(* CODESYS project Tc3_Mc3Ptp.library
   TcLibraryId: Beckhoff Automation GmbH|Tc3_Mc3Ptp|4.0.17.0
   Company: Beckhoff Automation GmbH
   Title: Tc3_Mc3Ptp
   Placeholder: Tc3_Mc3Ptp
   Version: 4.0.17.0

Project tree, tasks and I/O mapping:
  libraries: Tc3_Mc3Base, 4.0.17.0 (Beckhoff Automation GmbH)
  Motion Objects/
    function block AXIS_REF [ST]: FB_init, FB_exit, InitializeWithOid, GetCamming1DOid, GetPtpErrorResettableOid, GetErrorTriggerableOid, GetMaster1DOid, GetMotionObjectOid, GetPhasing1DOid, GetPtpReadWriteParameterOid, GetPtpSetPositionOid, GetPtpSetHomingStateOid, GetPtpTouchProbeOid, Name, Oid
    function block ENCODER_AXIS_REF [ST]: FB_init, FB_exit, GetPtpErrorResettableOid, GetErrorTriggerableOid, GetMaster1DOid, GetPtpReadWriteParameterOid, GetPtpSetPositionOid, GetPtpSetHomingStateOid, GetPtpTouchProbeOid, Name, Oid
    data type AXIS_REF_TOMC
    data type AXIS_REF_TOPLC
    data type ENCODER_AXIS_REF_TOPLC
  Administrative/
    function block MC_Reset [ST]: FB_init, FB_exit
    function block MC_Power [ST]: FB_init, FB_exit
    function block MC_SetOverride [ST]: FB_init, FB_exit
    Status/
      function block MC_ReadActualPosition [ST]: FB_init, FB_exit
      function block MC_ReadActualTorque [ST]: FB_init, FB_exit
      function block MC_ReadActualVelocity [ST]: FB_init, FB_exit
      function block MC_ReadAxisError [ST]: FB_init, FB_exit
      function block MC_ReadStatus [ST]: FB_init, FB_exit
    function block MC_SetPosition [ST]: FB_init, FB_exit
    Parameter/
      function block MC_WriteHardwareParameter [ST]: FB_init, FB_exit
      function block MC_ReadHardwareParameter [ST]: FB_init, FB_exit
      function block MC_ReadParameter [ST]: FB_init, FB_exit
      function block MC_WriteParameter [ST]: FB_init, FB_exit
      function block MC_ReadBoolParameter [ST]: FB_init, FB_exit
      function block MC_WriteBoolParameter [ST]: FB_init, FB_exit
      data type EAxisParameterId
      data type EReadMode
  External Setpoint Generator/
    function block MC_ActivateExternalSetpointGeneration [ST]: FB_init, FB_exit
    function block MC_ExternalSetpointGenerator [ST]: FB_init, FB_reinit, FB_exit, TcAddRef, TcQueryInterface, TcRelease, GetClassId, TcGetObjectId, TcGetObjectName, TcSetObjectId, TcSetObjectName, TcSetObjState, TcGetObjState, TcGetObjPara, TcSetObjPara, TcGetParentObjId, TcSetParentObjId, OnPreparation, OnStartPointInitialization, OnCyclicSetpointGeneration, OnDeactivation
  Discrete Motion/
    function block MC_Halt [ST]: FB_init, FB_exit
    function block MC_MoveAbsolute [ST]: FB_init, FB_exit
    function block MC_MoveModulo [ST]: FB_init, FB_exit
    function block MC_MoveRelative [ST]: FB_init, FB_exit
    function block MC_Stop [ST]: FB_init, FB_exit
    function block MC_WaitForStableActualPosition [ST]: FB_init, FB_exit
    data type EModuloDirection
  Synchronized Motion/
    function block MC_GearIn [ST]: FB_init, FB_exit
    function block MC_GearInPos [ST]: FB_init, FB_exit
    function block MC_PhasingAbsolute [ST]: FB_init, FB_exit
    function block MC_PhasingRelative [ST]: FB_init, FB_exit
    function block MC_HaltPhasing [ST]: FB_init, FB_exit
    data type EGearInPosSyncState
  Continuous Motion/
    function block MC_MoveVelocity [ST]: FB_init, FB_exit
    function block MC_Jog [ST]: FB_init, FB_exit
    data type EJogMode
  Homing/
    function block MC_SetHomingState [ST]: FB_init, FB_exit
    function block MC_Home [ST]: FB_init, FB_exit
    data type EHomingMode
  TouchProbe/
    function block MC_TouchProbe [ST]: FB_init, FB_exit
    function block MC_AbortTrigger [ST]: FB_init, FB_exit
    function block DriveTouchProbeRef [ST]: FB_init, FB_reinit, FB_exit
    function block EncoderTouchProbeRef [ST]: FB_init, FB_reinit, FB_exit
    function block TimestampTouchProbeRef [ST]: FB_init, FB_reinit, FB_exit
    function block BinaryTouchProbeRef [ST]: FB_init, FB_reinit, FB_exit
    function block FixedStopTouchProbeRef [ST]: FB_init, FB_reinit, FB_exit
    data type TouchProbeOptions
    data type ECoeTouchProbeInput
    data type CoeTouchProbeSettings
    data type FixedStopTouchProbeSettings
    data type EIncrementalEncoderTouchProbeSource
    data type IncrementalEncoderTouchProbeSettings
    data type TRIGGER_REF
    data type TouchProbeUnit
  Load Control/
    function block MC_LoadControl [ST]: FB_init, FB_exit
  Types/
    interface Type_PtpErrorResettable: GetPtpErrorResettableOid
    interface Type_PtpReadWriteParameter: GetPtpReadWriteParameterOid
    interface Type_PtpSetPosition: GetPtpSetPositionOid
    interface Type_PtpSetHomingState: GetPtpSetHomingStateOid
    interface Type_PtpTouchProbe: GetPtpTouchProbeOid
  DUTs/
    data type ESource
  Version/
    global variables Global_Version
*)

// Motion Objects/AXIS_REF_TOMC
(* Contains the information of the AXIS_REF passed from PLC to MC. *)
{attribute 'TcIecLibraryType'}
{attribute 'Namespace' := 'Tc3_Mc3Ptp'}
TYPE AXIS_REF_TOMC : 
	STRUCT
		(* Standard data from PLC to MC. *)
		{attribute 'GUID' := '928ACD6D-34F6-4728-BC12-CB3937EB34C2'}
		{attribute 'Namespace' := 'MC'}
		Std : MC.CDT_PLCTOMC_AXIS_STD;
	END_STRUCT
END_TYPE

// Motion Objects/AXIS_REF_TOPLC
(* Contains the information of the AXIS_REF passed from MC to PLC. *)
{attribute 'TcIecLibraryType'}
{attribute 'Namespace' := 'Tc3_Mc3Ptp'}
TYPE AXIS_REF_TOPLC : 
	STRUCT
		(* Reference to standard data from MC to PLC. *)
		{attribute 'TcPointerMapping'}
		{attribute 'GUID' := 'E7BFE865-900F-4F3A-B607-76F75FE96459'}
		{attribute 'Namespace' := 'MC'}
		Std : REFERENCE TO MC.CDT_MCTOPLC_AXIS_STD;
		(* Reference to setpoint data from MC *)
		{attribute 'TcPointerMapping'}
		{attribute 'GUID' := '0B0DBDAE-EDDB-492C-A6B1-EEFFED71DF0D'}
		{attribute 'Namespace' := 'MC'}
		Set : REFERENCE TO MC.CDT_MCTOPLC_AXIS_SET;
		(* Reference to actpoint data from MC *)
		{attribute 'TcPointerMapping'}
		{attribute 'GUID' := 'B6A63539-66D5-4BB4-8876-F4726B259807'}
		{attribute 'Namespace' := 'MC'}
		Act : REFERENCE TO MC.CDT_MCTOPLC_AXIS_ACT;
		 {attribute 'hide'}
		_reserved1 : ARRAY [1..4] OF UINT_8_16;
		(* Reference to modulo positions of a modulo axis *)
		{attribute 'TcPointerMapping'}
		{attribute 'GUID' := 'A44CE81F-76FF-4B9B-9906-BBAF0C1247D2'}
		{attribute 'Namespace' := 'MC'}
		Modulo : REFERENCE TO MC.CDT_MCTOPLC_AXIS_MODULO;
		(* Reference to loadcontrol data from MC *)
		{attribute 'TcPointerMapping'}
		{attribute 'GUID' := 'FAA1A803-EAD7-4A75-B851-39DA12582F94'}
		{attribute 'Namespace' := 'MC'}
		LoadControl : REFERENCE TO MC.CDT_MCTOPLC_AXIS_LOADCONTROL;
		 {attribute 'hide'}
		_reserved2 : ARRAY [1..8] OF UINT_8_16;
		(* Reference to fluidpower data from MC *)
		{attribute 'TcPointerMapping'}
		{attribute 'GUID' := 'ABD7A116-8AB9-4E1A-99C3-07858EE414A0'}
		{attribute 'Namespace' := 'MC'}
		FluidPower : REFERENCE TO MC.CDT_MCTOPLC_AXIS_FLUIDPOWER;
	END_STRUCT
END_TYPE

// Motion Objects/ENCODER_AXIS_REF_TOPLC
(* Contains the information of the ENCODER_AXIS_REF passed from MC to PLC. *)
{attribute 'TcIecLibraryType'}
{attribute 'Namespace' := 'Tc3_Mc3Ptp'}
TYPE ENCODER_AXIS_REF_TOPLC : 
	STRUCT
		(* Reference to standard data from MC to PLC. *)
		{attribute 'TcPointerMapping'}
		{attribute 'GUID' := 'B8555454-C37F-461B-AA7A-1853577E270C'}
		{attribute 'Namespace' := 'MC'}
		Std : REFERENCE TO MC.CDT_MCTOPLC_ENCODER_AXIS_STD;
		(* Reference to actual data from MC. *)
		{attribute 'TcPointerMapping'}
		{attribute 'GUID' := '104567DA-4469-4052-8B31-85248F22B6DF'}
		{attribute 'Namespace' := 'MC'}
		Act : REFERENCE TO MC.CDT_MCTOPLC_ENCODER_AXIS_ACT;
		(* Reference to modulo positions from encoder axis. *)
		{attribute 'TcPointerMapping'}
		{attribute 'GUID' := '7B38ABBA-E075-4ACD-87B2-5F73D822C5F9'}
		{attribute 'Namespace' := 'MC'}
		Modulo : REFERENCE TO MC.CDT_MCTOPLC_ENCODER_AXIS_MODULO;
	END_STRUCT
END_TYPE

// Discrete Motion/EModuloDirection
(* Direction of travel for modulo positioning. *)
{attribute 'TcIecLibraryType'}
{attribute 'Namespace' := 'Tc3_Mc3Ptp'}
{attribute 'strict'}
{attribute 'qualified_only'}
{attribute 'to_string'}
TYPE EModuloDirection : (
	ShortestDistance:=0, 	(* Move in the direction that results in the shortest travel distance. *)
	PositiveDirection:=1, 	(* Always move in the positive direction to reach the target. *)
	NegativeDirection:=2	(* Always move in the negative direction to reach the target. *)
) UINT;
END_TYPE

// Synchronized Motion/EGearInPosSyncState
(* Synchronization state reported by MC_GearInPos for the PhysicalAxis. Combines whether the slave is synchronized to the master with whether the master has already passed its master sync position. Reports 'Waiting' while the slave cannot move yet due to a sync direction restriction. *)
{attribute 'TcIecLibraryType'}
{attribute 'Namespace' := 'Tc3_Mc3Ptp'}
{attribute 'strict'}
{attribute 'qualified_only'}
{attribute 'to_string'}
TYPE EGearInPosSyncState : (
	Invalid:=0, 	(* Default value before the function block has been activated. *)
	Waiting:=1, 	(* The slave cannot start to move yet because the master is moving against the restricted sync direction. *)
	Synchronizing:=2, 	(* The synchronization is not yet complete and the master has not yet passed its master sync position. *)
	SynchronizingAfterMasterSyncPosition:=3, 	(* The synchronization is not yet complete; the master has already passed its master sync position. *)
	InSyncBeforeMasterSyncPosition:=4, 	(* The slave is locked in to the master, but the master has not yet passed its master sync position. *)
	InSync:=5	(* The slave is locked in to the master and the master has passed its master sync position. *)
) UDINT;
END_TYPE

// Continuous Motion/EJogMode
(* Selects the jog operation mode. *)
{attribute 'TcIecLibraryType'}
{attribute 'Namespace' := 'Tc3_Mc3Ptp'}
{attribute 'strict'}
{attribute 'qualified_only'}
{attribute 'to_string'}
TYPE EJogMode : (
	StandardSlow:=1, 	(* Jog at low velocity using the configured slow jog speed. *)
	StandardFast:=2, 	(* Jog at high velocity using the configured fast jog speed. *)
	Continuous:=3, 	(* Jog continuously at the commanded velocity while the jog input is active. *)
	Inching:=4	(* Move a fixed incremental distance for each jog activation. *)
) UINT;
END_TYPE

// Homing/EHomingMode
(* Mode selection for functional configuration of MC_SetHomingState command. *)
{attribute 'TcIecLibraryType'}
{attribute 'Namespace' := 'Tc3_Mc3Ptp'}
{attribute 'qualified_only'}
{attribute 'strict'}
{attribute 'to_string'}
TYPE EHomingMode : (
	ForceIsHomed:=0, 	(* Sets the homing state to homed (IsPositionValid = TRUE) without performing any movement or position change. *)
	ResetIsHomed:=1, 	(* Resets the homing state to not homed (IsPositionValid = FALSE). *)
	ForceIsHomedAtPosition:=2	(* Sets the current position to the specified homing position and marks the axis as homed (IsPositionValid = TRUE). *)
) UDINT;
END_TYPE

// TouchProbe/TouchProbeOptions
(* MC_TouchProbe Options *)
{attribute 'TcIecLibraryType'}
{attribute 'Namespace' := 'Tc3_Mc3Ptp'}
TYPE TouchProbeOptions : 
	STRUCT
		(* Start position from where trigger events are accepted ([PosUnit], included in the position window).
		It can be left as 'Ignore' if no lower limit is desired. Must have value <= WindowLastPosition otherwise. *)
		WindowFirstPosition : LREAL := STRING_TO_LREAL('#Ignore');
		(* Stop position up to where trigger events are accepted ([PosUnit], included in the position window).
		It can be left as 'Ignore' if no upper limit is desired. Must have value >= WindowFirstPosition otherwise.
		 *)
		WindowLastPosition : LREAL := STRING_TO_LREAL('#Ignore');
		(* Calculate RecordedPosition as modulo value. *)
		PositionsAsModuloValues : BOOL := false;
		(* Continuous recording mode *)
		Continuous : BOOL := false;
		 {attribute 'hide'}
		_reserved1 : ARRAY [1..6] OF USINT;
	END_STRUCT
END_TYPE

// TouchProbe/ECoeTouchProbeInput
(* Selection for CoE Drive touch probe input. *)
{attribute 'TcIecLibraryType'}
{attribute 'Namespace' := 'Tc3_Mc3Ptp'}
{attribute 'qualified_only'}
{attribute 'strict'}
{attribute 'to_string'}
TYPE ECoeTouchProbeInput : (
	DriveDefault:=0, 	(* Trigger on the touch probe default input (i.e., the digital input 1/2 mapped to TouchProbe1/TouchProbe2 functionality in the drive). *)
	ZeroImpulse:=1, 	(* Trigger on the main encoder index signal (encoder Z/index). Only valid if the drive exposes the index signal to the touch probe function. *)
	DriveDefined:=2, 	(* Trigger source is defined by object 0x60D0/0x8001 (DS402/MDP742). *)
	ConfiguredInAxis:=255	(* The touch probe input source is configured in the axis (TCOM object). The value specified at the CoeDriveSettings input is ignored. *)
) UDINT;
END_TYPE

// TouchProbe/CoeTouchProbeSettings
(* CoE drive-specific touch probe source settings. *)
{attribute 'TcIecLibraryType'}
{attribute 'Namespace' := 'Tc3_Mc3Ptp'}
TYPE CoeTouchProbeSettings : 
	STRUCT
		(* Input source for touch probe 1. *)
		{attribute 'GUID' := '119F1828-69D6-4F12-9086-EF2FF951D8CC'}
		{attribute 'Namespace' := 'Tc3_Mc3Ptp'}
		TouchProbe1Source : ECoeTouchProbeInput := ECoeTouchProbeInput.ConfiguredInAxis;
		(* Input source for touch probe 2. *)
		{attribute 'GUID' := '119F1828-69D6-4F12-9086-EF2FF951D8CC'}
		{attribute 'Namespace' := 'Tc3_Mc3Ptp'}
		TouchProbe2Source : ECoeTouchProbeInput := ECoeTouchProbeInput.ConfiguredInAxis;
	END_STRUCT
END_TYPE

// TouchProbe/FixedStopTouchProbeSettings
(* Configure up to three thresholds for fixed stop detection (Torque, Velocity, Lag). Enter #Default to use the axis default value, or #Ignore to disable a threshold.
Typical detection criteria: combination of high torque, low velocity, and/or increasing lag. *)
{attribute 'TcIecLibraryType'}
{attribute 'Namespace' := 'Tc3_Mc3Ptp'}
TYPE FixedStopTouchProbeSettings : 
	STRUCT
		(* Threshold for the actual motor torque. If the torque exceeds this value during evaluation, it contributes to a fixed stop decision. Enter #Ignore to disable this threshold. *)
		TorqueThreshold : LREAL := STRING_TO_LREAL('#Default');
		(* Upper limit for the actual axis velocity during evaluation. Fixed stop detection is evaluated only while the absolute velocity is below this value. Enter #Ignore to disable this threshold. *)
		VelocityThreshold : LREAL := STRING_TO_LREAL('#Default');
		(* Threshold for the position following error (command position minus actual position). If the absolute following error exceeds this value during evaluation, it contributes to a fixed stop decision. Enter #Ignore to disable this threshold. *)
		LagThreshold : LREAL := STRING_TO_LREAL('#Default');
	END_STRUCT
END_TYPE

// TouchProbe/EIncrementalEncoderTouchProbeSource
(* Selection for incremental encoder touch probe latch source. *)
{attribute 'TcIecLibraryType'}
{attribute 'Namespace' := 'Tc3_Mc3Ptp'}
{attribute 'qualified_only'}
{attribute 'strict'}
{attribute 'to_string'}
TYPE EIncrementalEncoderTouchProbeSource : (
	LatchC:=0, 	(* Internal latch (encoder C-track / index signal). *)
	LatchExternPositive:=1, 	(* External latch input, capture on rising edge. *)
	LatchExternNegative:=2, 	(* External latch input, capture on falling edge. *)
	ConfiguredInAxis:=255	(* The touch probe latch source is configured in the axis (TCOM object). The value specified at the IncrementalEncoderSettings input is ignored. *)
) UDINT;
END_TYPE

// TouchProbe/IncrementalEncoderTouchProbeSettings
(* Touch probe settings for incremental encoder terminals. *)
{attribute 'TcIecLibraryType'}
{attribute 'Namespace' := 'Tc3_Mc3Ptp'}
TYPE IncrementalEncoderTouchProbeSettings : 
	STRUCT
		(* Latch source override for position capture. *)
		{attribute 'GUID' := 'B9DA70FA-AB67-491F-BE82-1393AA92E6AD'}
		{attribute 'Namespace' := 'Tc3_Mc3Ptp'}
		Source : EIncrementalEncoderTouchProbeSource := EIncrementalEncoderTouchProbeSource.ConfiguredInAxis;
	END_STRUCT
END_TYPE

// TouchProbe/TRIGGER_REF
{attribute 'TcIecLibraryType'}
{attribute 'Namespace' := 'Tc3_Mc3Ptp'}
{attribute 'hide'}
TYPE TRIGGER_REF : 
	STRUCT
		Target : UDINT;
		ProbeId : UINT;
		 {attribute 'hide'}
		_reserved1 : UINT;
		Edge : UDINT;
		 {attribute 'hide'}
		_reserved2 : UDINT;
		{attribute 'GUID' := '18071995-0000-0000-0000-000000000018'}
		ObjId : GLOBAL.PVOID;
		{attribute 'GUID' := '18071995-0000-0000-0000-000000000018'}
		SettingsCoe : GLOBAL.PVOID;
		{attribute 'GUID' := '18071995-0000-0000-0000-000000000018'}
		SettingsFixedStop : GLOBAL.PVOID;
		{attribute 'GUID' := '18071995-0000-0000-0000-000000000018'}
		SettingsIncrementalEncoder : GLOBAL.PVOID;
	END_STRUCT
END_TYPE

// TouchProbe/TouchProbeUnit
(* Contains trigger references for positive and negative edge touch probes. *)
{attribute 'TcIecLibraryType'}
{attribute 'Namespace' := 'Tc3_Mc3Ptp'}
TYPE TouchProbeUnit : 
	STRUCT
		(* Trigger reference for positive edge events. *)
		{attribute 'GUID' := 'CC3262A1-A7A1-46D3-802E-9117404E77E7'}
		{attribute 'Namespace' := 'Tc3_Mc3Ptp'}
		PositiveTrigger : TRIGGER_REF;
		(* Trigger reference for negative edge events. *)
		{attribute 'GUID' := 'CC3262A1-A7A1-46D3-802E-9117404E77E7'}
		{attribute 'Namespace' := 'Tc3_Mc3Ptp'}
		NegativeTrigger : TRIGGER_REF;
	END_STRUCT
END_TYPE

// DUTs/ESource
(* Selects between setpoint and actual value as data source. *)
{attribute 'TcIecLibraryType'}
{attribute 'Namespace' := 'Tc3_Mc3Ptp'}
{attribute 'hide'}
{attribute 'to_string'}
TYPE ESource : (
	SetValue:=0, 	(* Use the commanded setpoint value. *)
	ActualValue:=1	(* Use the measured actual value from the encoder. *)
) UINT;
END_TYPE

// Administrative/Parameter/EAxisParameterId
(* Parameter IDs for reading and writing axis parameters via MC_ReadParameter / MC_WriteParameter (MC_ReadBoolParameter / MC_WriteBoolParameter). *)
{attribute 'TcIecLibraryType'}
{attribute 'Namespace' := 'Tc3_Mc3Ptp'}
{attribute 'strict'}
{attribute 'qualified_only'}
{attribute 'to_string'}
TYPE EAxisParameterId : (
	Invalid:=16#0000000000000000, 
	MaximumVelocity:=16#0000000005093009, 	(* Use MC_ReadParameter, MC_WriteParameter *)
	MaximumAcceleration:=16#000000000509300a, 	(* Use MC_ReadParameter, MC_WriteParameter *)
	MaximumDeceleration:=16#000000000509300b, 	(* Use MC_ReadParameter, MC_WriteParameter *)
	DefaultAcceleration:=16#000000000509300c, 	(* Use MC_ReadParameter, MC_WriteParameter *)
	DefaultDeceleration:=16#000000000509300d, 	(* Use MC_ReadParameter, MC_WriteParameter *)
	DefaultJerk:=16#000000000509300e, 	(* Use MC_ReadParameter, MC_WriteParameter *)
	MaximumJerk:=16#0000000005093015, 	(* Use MC_ReadParameter, MC_WriteParameter *)
	MinimumPosition:=16#0000000005093021, 	(* Use MC_ReadParameter, MC_WriteParameter *)
	MaximumPosition:=16#0000000005093023, 	(* Use MC_ReadParameter, MC_WriteParameter *)
	PositionModulus:=16#0000000005030107, 	(* Use MC_ReadParameter, MC_WriteParameter *)
	PositionModuloToleranceWindow:=16#0000000005030108, 	(* Use MC_ReadParameter, MC_WriteParameter *)
	MaximumPositionLagValue:=16#000000000503011b, 	(* Use MC_ReadParameter, MC_WriteParameter *)
	MaximumPositionLagFilterTime:=16#000000000503011c, 	(* Use MC_ReadParameter, MC_WriteParameter *)
	JogVelocitySlow:=16#000000000503019e, 	(* Use MC_ReadParameter, MC_WriteParameter *)
	JogVelocityFast:=16#000000000503019f, 	(* Use MC_ReadParameter, MC_WriteParameter *)
	MinimumPositionLag:=16#00000000050301a1, 	(* Use MC_ReadParameter, MC_WriteParameter *)
	MaximumPositionLag:=16#00000000050301a2, 	(* Use MC_ReadParameter, MC_WriteParameter *)
	VelocityOverrideFactor:=16#0000000005030231, 	(* Use MC_ReadParameter, MC_WriteParameter *)
	SimulationMode:=16#00000000050300b1, 	(* Use MC_ReadBoolParameter, MC_WriteBoolParameter *)
	IsModuloAxis:=16#0000000005030101, 	(* Use MC_ReadBoolParameter, MC_WriteBoolParameter *)
	PositionLagMonitoringEnabled:=16#000000000503011a, 	(* Use MC_ReadBoolParameter, MC_WriteBoolParameter *)
	PositionLimitEnforcementEnabled:=16#000000000503015d, 	(* Use MC_ReadBoolParameter, MC_WriteBoolParameter *)
	DriveVelocityScalingNumeratorToHardware:=16#0000000105030122, 	(* Use MC_ReadParameter, MC_WriteParameter *)
	DriveVelocityScalingDenominatorToHardware:=16#00000001050301a7, 	(* Use MC_ReadParameter, MC_WriteParameter *)
	DriveTorqueScalingFromHardware:=16#000000010503014f, 	(* Use MC_ReadParameter, MC_WriteParameter *)
	DriveTimeoutForEnableAndReset:=16#000000010503d004, 	(* Use MC_ReadParameter, MC_WriteParameter *)
	DriveActiveHomingOffset:=16#0000000105030224, 	(* Use MC_ReadParameter, MC_WriteParameter *)
	DriveDirectionInverted:=16#00000001050301b2, 	(* Use MC_ReadBoolParameter, MC_WriteBoolParameter *)
	EncoderPositionScalingNumeratorFromHardware:=16#0000000205030103, 	(* Use MC_ReadParameter, MC_WriteParameter *)
	EncoderPositionScalingDenominatorFromHardware:=16#0000000205030104, 	(* Use MC_ReadParameter, MC_WriteParameter *)
	EncoderMountingOffset:=16#0000000205030106, 	(* Use MC_ReadParameter, MC_WriteParameter *)
	EncoderWorkZeroOffset:=16#00000002050301d1, 	(* Use MC_ReadParameter, MC_WriteParameter *)
	EncoderDirectionInverted:=16#00000002050301b2, 	(* Use MC_ReadBoolParameter, MC_WriteBoolParameter *)
	EncoderIsHomed:=16#000000020503d070, 	(* Use MC_ReadBoolParameter, MC_WriteBoolParameter *)
	EncoderIsAbsolutePositionValid:=16#000000020503d071	(* Use MC_ReadBoolParameter, MC_WriteBoolParameter *)
) ULINT;
END_TYPE

// Administrative/Parameter/EReadMode
(* Selects the read operation mode. *)
{attribute 'TcIecLibraryType'}
{attribute 'Namespace' := 'Tc3_Mc3Ptp'}
{attribute 'strict'}
{attribute 'qualified_only'}
{attribute 'to_string'}
TYPE EReadMode : (
	Once:=1, 	(* Read the parameter value once. *)
	Cyclic:=2	(* Read the parameter value cyclically. *)
) UDINT;
END_TYPE

// Version/Global_Version
{attribute 'TcGenerated'}
// This function has been automatically generated from the project information.
VAR_GLOBAL CONSTANT
	{attribute 'const_non_replaced'}
	{attribute 'linkalways'}
	stLibVersion_Tc3_Mc3Ptp : ST_LibVersion := (iMajor := 4, iMinor := 0, iBuild := 17, iRevision := 0, nFlags := 0, sVersion := '4.0.17.0');
	{attribute 'const_non_replaced'}
	{attribute 'linkalways'}
	sLibraryId_Tc3_Mc3Ptp : String := 'Beckhoff Automation GmbH|Tc3_Mc3Ptp|4.0.17.0';
END_VAR

// Motion Objects/AXIS_REF

{attribute 'c++_compatible'}
{attribute 'external_name' := 'AXIS_REF_GUID_931209B0_6FAC_E9BE_F824_23CE2FAA5732'}
{attribute 'TcIecLibraryType'}
(* 
        An MC3 axis used with PLCopen motion control function blocks.
	 *)
FUNCTION_BLOCK AXIS_REF IMPLEMENTS Tc3_Mc3Base.Type_Camming1D, Type_PtpErrorResettable, Tc3_Mc3Base.Type_ErrorTriggerable, Tc3_Mc3Base.Type_Master1D, Tc3_Mc3Base.Type_MotionObject, Tc3_Mc3Base.Type_Phasing1D, Type_PtpReadWriteParameter, Type_PtpSetPosition, Type_PtpSetHomingState, Type_PtpTouchProbe
VAR
END_VAR
VAR_INPUT
	(* Data area for cyclic PLC-to-MC data exchange (mapped to MC axis TcCOM object input process image). *)
	{attribute 'GUID' := '70EBE612-C6D0-4BB5-85F1-59AB9BBF86DE'}
	{attribute 'Namespace' := 'Tc3_Mc3Ptp'}
	PlcToMc AT %Q* : AXIS_REF_TOMC;
	(* Data area for cyclic MC-to-PLC data exchange (mapped to MC axis TcCOM object output process image). *)
	{attribute 'GUID' := '99E83C85-C326-4077-86A5-05990B8F1158'}
	{attribute 'Namespace' := 'Tc3_Mc3Ptp'}
	McToPlc AT %I* : AXIS_REF_TOPLC;
END_VAR
VAR
	{attribute 'hide'}
	_reserved : UDINT;
	 {attribute 'hide'}
	_reserved1 : UINT_0_32;
END_VAR

{attribute 'TcTypeSystem'}

(* Internal method *)
{attribute 'hide'}
METHOD FB_init : BOOL
VAR_INPUT
	(*  if TRUE, the retain variables are initialized (warm start / cold start) *)
	bInitRetains : BOOL;
	(*  if TRUE, the instance afterwards gets moved into the copy code (online change) *)
	bInCopyCode : BOOL;
END_VAR
END_METHOD

{attribute 'TcTypeSystem'}

(* Internal method *)
{attribute 'hide'}
METHOD FB_exit : BOOL
VAR_INPUT
	(*  if TRUE, the exit method is called for exiting an instance that is copied afterwards (online change). *)
	bInCopyCode : BOOL;
END_VAR
END_METHOD

{attribute 'TcTypeSystem'}

(* Internal method to wrap object ID *)
{attribute 'hide'}
METHOD InitializeWithOid
VAR_INPUT
	(* Object ID which is used as an alternative when this is used as master. *)
	{attribute 'GUID' := '18071995-0000-0000-0000-00000000000F'}
	NewOid : GLOBAL.OTCID;
END_VAR
END_METHOD

{attribute 'TcTypeSystem'}

{attribute 'c++_external'}
{attribute 'hide'}
METHOD GetCamming1DOid : GLOBAL.OTCID
END_METHOD

{attribute 'TcTypeSystem'}

{attribute 'c++_external'}
{attribute 'hide'}
METHOD GetPtpErrorResettableOid : GLOBAL.OTCID
END_METHOD

{attribute 'TcTypeSystem'}

{attribute 'c++_external'}
{attribute 'hide'}
METHOD GetErrorTriggerableOid : GLOBAL.OTCID
END_METHOD

{attribute 'TcTypeSystem'}

{attribute 'c++_external'}
{attribute 'hide'}
METHOD GetMaster1DOid : GLOBAL.OTCID
END_METHOD

{attribute 'TcTypeSystem'}

{attribute 'c++_external'}
{attribute 'hide'}
METHOD GetMotionObjectOid : GLOBAL.OTCID
END_METHOD

{attribute 'TcTypeSystem'}

{attribute 'c++_external'}
{attribute 'hide'}
METHOD GetPhasing1DOid : GLOBAL.OTCID
END_METHOD

{attribute 'TcTypeSystem'}

{attribute 'c++_external'}
{attribute 'hide'}
METHOD GetPtpReadWriteParameterOid : GLOBAL.OTCID
END_METHOD

{attribute 'TcTypeSystem'}

{attribute 'c++_external'}
{attribute 'hide'}
METHOD GetPtpSetPositionOid : GLOBAL.OTCID
END_METHOD

{attribute 'TcTypeSystem'}

{attribute 'c++_external'}
{attribute 'hide'}
METHOD GetPtpSetHomingStateOid : GLOBAL.OTCID
END_METHOD

{attribute 'TcTypeSystem'}

{attribute 'c++_external'}
{attribute 'hide'}
METHOD GetPtpTouchProbeOid : GLOBAL.OTCID
END_METHOD

{attribute 'TcTypeSystem'}

	(* Returns the configured name of the axis. *)
{attribute 'monitoring' := 'call'}
	PROPERTY Name : STRING(255)
GET
END_GET
END_PROPERTY

{attribute 'TcTypeSystem'}

	(* Returns the TcCOM object ID of the axis. *)
{attribute 'monitoring' := 'call'}
	PROPERTY Oid : GLOBAL.OTCID
GET
END_GET
END_PROPERTY

END_FUNCTION_BLOCK

// Types/Type_PtpErrorResettable
(* Type for a motion control object whose errors can be reset (e. g. supported by AXIS_REF). *)
{attribute 'Namespace' := 'Tc3_Mc3Ptp'}
{attribute 'c++_compatible'}
INTERFACE Type_PtpErrorResettable

{attribute 'TcTypeSystem'}
{attribute 'c++_compatible'}
{attribute 'minimal_input_size' := '4'}
{attribute 'pack_mode' := '4'}
{attribute 'hide'}
METHOD GetPtpErrorResettableOid : GLOBAL.OTCID
END_METHOD

END_INTERFACE

// Types/Type_PtpReadWriteParameter
(* Type for a motion control object that supports parameter read/write access (e.g. supported by AXIS_REF and ENCODER_AXIS_REF). *)
{attribute 'Namespace' := 'Tc3_Mc3Ptp'}
{attribute 'c++_compatible'}
INTERFACE Type_PtpReadWriteParameter

{attribute 'TcTypeSystem'}
{attribute 'c++_compatible'}
{attribute 'minimal_input_size' := '4'}
{attribute 'pack_mode' := '4'}
{attribute 'hide'}
METHOD GetPtpReadWriteParameterOid : GLOBAL.OTCID
END_METHOD

END_INTERFACE

// Motion Objects/ENCODER_AXIS_REF

{attribute 'c++_compatible'}
{attribute 'external_name' := 'ENCODER_AXIS_REF_GUID_E0F25744_2FAD_E888_F942_A6877B2D0404'}
{attribute 'TcIecLibraryType'}
(* 
        An MC3 encoder axis used with PLCopen motion control function blocks.
	 *)
FUNCTION_BLOCK ENCODER_AXIS_REF IMPLEMENTS Type_PtpErrorResettable, Tc3_Mc3Base.Type_ErrorTriggerable, Tc3_Mc3Base.Type_Master1D, Type_PtpReadWriteParameter, Type_PtpSetPosition, Type_PtpSetHomingState, Type_PtpTouchProbe
VAR
END_VAR
VAR_INPUT
	(* Data area for cyclic MC-to-PLC data exchange (mapped to MC encoder axis TcCOM object output process image). *)
	{attribute 'GUID' := 'B5C6D7E8-F9A0-4B1C-2D3E-4F5A6B7C8D9E'}
	{attribute 'Namespace' := 'Tc3_Mc3Ptp'}
	McToPlc AT %I* : ENCODER_AXIS_REF_TOPLC;
END_VAR

{attribute 'TcTypeSystem'}

(* Internal method *)
{attribute 'hide'}
METHOD FB_init : BOOL
VAR_INPUT
	(*  if TRUE, the retain variables are initialized (warm start / cold start) *)
	bInitRetains : BOOL;
	(*  if TRUE, the instance afterwards gets moved into the copy code (online change) *)
	bInCopyCode : BOOL;
END_VAR
END_METHOD

{attribute 'TcTypeSystem'}

(* Internal method *)
{attribute 'hide'}
METHOD FB_exit : BOOL
VAR_INPUT
	(*  if TRUE, the exit method is called for exiting an instance that is copied afterwards (online change). *)
	bInCopyCode : BOOL;
END_VAR
END_METHOD

{attribute 'TcTypeSystem'}

{attribute 'c++_external'}
{attribute 'hide'}
METHOD GetPtpErrorResettableOid : GLOBAL.OTCID
END_METHOD

{attribute 'TcTypeSystem'}

{attribute 'c++_external'}
{attribute 'hide'}
METHOD GetErrorTriggerableOid : GLOBAL.OTCID
END_METHOD

{attribute 'TcTypeSystem'}

{attribute 'c++_external'}
{attribute 'hide'}
METHOD GetMaster1DOid : GLOBAL.OTCID
END_METHOD

{attribute 'TcTypeSystem'}

{attribute 'c++_external'}
{attribute 'hide'}
METHOD GetPtpReadWriteParameterOid : GLOBAL.OTCID
END_METHOD

{attribute 'TcTypeSystem'}

{attribute 'c++_external'}
{attribute 'hide'}
METHOD GetPtpSetPositionOid : GLOBAL.OTCID
END_METHOD

{attribute 'TcTypeSystem'}

{attribute 'c++_external'}
{attribute 'hide'}
METHOD GetPtpSetHomingStateOid : GLOBAL.OTCID
END_METHOD

{attribute 'TcTypeSystem'}

{attribute 'c++_external'}
{attribute 'hide'}
METHOD GetPtpTouchProbeOid : GLOBAL.OTCID
END_METHOD

{attribute 'TcTypeSystem'}

	(* Returns the configured name of the encoder axis. *)
{attribute 'monitoring' := 'call'}
	PROPERTY Name : STRING(255)
GET
END_GET
END_PROPERTY

{attribute 'TcTypeSystem'}

	(* Returns the TcCOM object ID of the encoder axis. *)
{attribute 'monitoring' := 'call'}
	PROPERTY Oid : GLOBAL.OTCID
GET
END_GET
END_PROPERTY

END_FUNCTION_BLOCK

// Types/Type_PtpSetPosition
(* Type for a motion control object that supports setting position (e. g. supported by AXIS_REF). *)
{attribute 'Namespace' := 'Tc3_Mc3Ptp'}
{attribute 'c++_compatible'}
INTERFACE Type_PtpSetPosition

{attribute 'TcTypeSystem'}
{attribute 'c++_compatible'}
{attribute 'minimal_input_size' := '4'}
{attribute 'pack_mode' := '4'}
{attribute 'hide'}
METHOD GetPtpSetPositionOid : GLOBAL.OTCID
END_METHOD

END_INTERFACE

// Types/Type_PtpSetHomingState
(* Type for a motion control object that supports setting the homing state (e. g. supported by AXIS_REF and ENCODER_AXIS_REF). *)
{attribute 'Namespace' := 'Tc3_Mc3Ptp'}
{attribute 'c++_compatible'}
INTERFACE Type_PtpSetHomingState

{attribute 'TcTypeSystem'}
{attribute 'c++_compatible'}
{attribute 'minimal_input_size' := '4'}
{attribute 'pack_mode' := '4'}
{attribute 'hide'}
METHOD GetPtpSetHomingStateOid : GLOBAL.OTCID
END_METHOD

END_INTERFACE

// Types/Type_PtpTouchProbe
(* Type for a motion control object that supports touch probe commands (e. g. supported by AXIS_REF and ENCODER_AXIS_REF). *)
{attribute 'Namespace' := 'Tc3_Mc3Ptp'}
{attribute 'c++_compatible'}
INTERFACE Type_PtpTouchProbe

{attribute 'TcTypeSystem'}
{attribute 'c++_compatible'}
{attribute 'minimal_input_size' := '4'}
{attribute 'pack_mode' := '4'}
{attribute 'hide'}
METHOD GetPtpTouchProbeOid : GLOBAL.OTCID
END_METHOD

END_INTERFACE

// Administrative/MC_Reset

{attribute 'c++_compatible'}
{attribute 'external_name' := 'MC_Reset_GUID_C09B70BA_4675_EE3C_E76C_41428371BC38'}
{attribute 'TcIecLibraryType'}
{attribute 'hide_all_locals'}
(* 
		This function block resets all motion object-related errors and transitions the motion object out of state ErrorStop.<br/>
		The resulting state is Disabled, if no Enable is requested for the motion object (e.g. via MC_Power).<br/>
		It results in DiscreteMotion, if the motion object has a closed control loop and a controlled error reaction is still ongoing.<br/>
		Otherwise, Standstill is the resulting state. This function block does not affect the output of motion function block instances.
	 *)
FUNCTION_BLOCK MC_Reset
VAR_INPUT
	(* Interface pointer to the object on which the command should be performed (e.g. Axis, Linear Mover). *)
	{attribute 'GUID' := '871876B3-D74D-4115-B995-E302FD1B35FF'}
	{attribute 'Namespace' := 'Tc3_Mc3Ptp'}
	Axis : Type_PtpErrorResettable;
	(* Trigger the command with rising edge. *)
	Execute : BOOL;
END_VAR
VAR_OUTPUT
	(* Potential axis and/or drive error has been reset. State Standstill, Disabled or DiscreteMotion is reached. *)
	Done : BOOL;
	(* Function block is not finished and new output values are to be expected. *)
	Busy : BOOL;
	(* Error occurred within function block. *)
	Error : BOOL;
	(* Error identifier *)
	ErrorId : UDINT;
END_VAR
VAR
	 {attribute 'hide'}
	_reserved1 : UINT_0_32;
	 {attribute 'hide'}
	_reserved2 : ARRAY [1..20] OF UINT_8_16;
	 {attribute 'hide'}
	_reserved3 : ARRAY [1..28] OF USINT;
END_VAR

{attribute 'TcTypeSystem'}

(* Internal method *)
{attribute 'hide'}
METHOD FB_init : BOOL
VAR_INPUT
	(*  if TRUE, the retain variables are initialized (warm start / cold start) *)
	bInitRetains : BOOL;
	(*  if TRUE, the instance afterwards gets moved into the copy code (online change) *)
	bInCopyCode : BOOL;
END_VAR
END_METHOD

{attribute 'TcTypeSystem'}

(* Internal method *)
{attribute 'hide'}
METHOD FB_exit : BOOL
VAR_INPUT
	(*  if TRUE, the exit method is called for exiting an instance that is copied afterwards (online change). *)
	bInCopyCode : BOOL;
END_VAR
END_METHOD

END_FUNCTION_BLOCK

// Administrative/MC_Power

{attribute 'c++_compatible'}
{attribute 'external_name' := 'MC_Power_GUID_DFCA01AC_8B4E_E5B3_DB59_8C7638CFE540'}
{attribute 'TcIecLibraryType'}
{attribute 'hide_all_locals'}
(* 
		This function block controls the power stage (on or off).
	 *)
FUNCTION_BLOCK MC_Power
VAR_IN_OUT
	(* Reference to the axis *)
	{attribute 'GUID' := '931209B0-6FAC-E9BE-F824-23CE2FAA5732'}
	{attribute 'Namespace' := 'Tc3_Mc3Ptp'}
	Axis : AXIS_REF;
END_VAR
VAR_INPUT
	(* General software enable for the axis *)
	Enable : BOOL;
	(* Feed enable in positive direction. Only effective if Enable = TRUE *)
	EnablePositive : BOOL := false;
	(* Feed enable in negative direction. Only effective if Enable = TRUE *)
	EnableNegative : BOOL := false;
END_VAR
VAR_OUTPUT
	(* Axis is ready for motion commands. *)
	Status : BOOL;
	(* Error occurred within function block or axis already signaling an error. *)
	Error : BOOL;
END_VAR
VAR
	 {attribute 'hide'}
	_reserved1 : ARRAY [1..3] OF USINT;
END_VAR
VAR_OUTPUT
	(* Error identifier of function block or axis *)
	ErrorId : UDINT;
END_VAR
VAR
	 {attribute 'hide'}
	_reserved2 : UINT_0_32;
END_VAR

{attribute 'TcTypeSystem'}

(* Internal method *)
{attribute 'hide'}
METHOD FB_init : BOOL
VAR_INPUT
	(*  if TRUE, the retain variables are initialized (warm start / cold start) *)
	bInitRetains : BOOL;
	(*  if TRUE, the instance afterwards gets moved into the copy code (online change) *)
	bInCopyCode : BOOL;
END_VAR
END_METHOD

{attribute 'TcTypeSystem'}

(* Internal method *)
{attribute 'hide'}
METHOD FB_exit : BOOL
VAR_INPUT
	(*  if TRUE, the exit method is called for exiting an instance that is copied afterwards (online change). *)
	bInCopyCode : BOOL;
END_VAR
END_METHOD

END_FUNCTION_BLOCK

// Administrative/MC_SetOverride

{attribute 'c++_compatible'}
{attribute 'external_name' := 'MC_SetOverride_GUID_EC43C2CD_0650_E2EE_F82C_55B33981EAD6'}
{attribute 'TcIecLibraryType'}
{attribute 'hide_all_locals'}
(* 
	This function block sets the velocity override factor that is applied to movement commands of the axis.
	The override factor does not apply to movement in the synchronized motion state (e.g. movement induced by MC_GearIn, MC_GearInPos, ...).
	 *)
FUNCTION_BLOCK MC_SetOverride
VAR_IN_OUT
	(* Reference to the axis *)
	{attribute 'GUID' := '931209B0-6FAC-E9BE-F824-23CE2FAA5732'}
	{attribute 'Namespace' := 'Tc3_Mc3Ptp'}
	Axis : AXIS_REF;
END_VAR
VAR_INPUT
	(* Write the velocity override factor continuously while Enable = TRUE. *)
	Enable : BOOL;
END_VAR
VAR
	 {attribute 'hide'}
	_reserved1 : ARRAY [1..7] OF USINT;
END_VAR
VAR_INPUT
	(* Applies to commanded velocities. Valid range is [0,1]. Use STRING_TO_LREAL('#Ignore') to NOT overwrite the previous value. *)
	VelocityFactor : LREAL := 1.0;
END_VAR
VAR
	 {attribute 'hide'}
	_reserved2 : ARRAY [1..8] OF USINT;
END_VAR
VAR_OUTPUT
	(* The commanded override is set. *)
	Enabled : BOOL;
	(* Error occurred within function block. *)
	Error : BOOL;
END_VAR
VAR
	 {attribute 'hide'}
	_reserved3 : UINT;
END_VAR
VAR_OUTPUT
	(* Error identifier *)
	ErrorId : UDINT;
END_VAR

{attribute 'TcTypeSystem'}

(* Internal method *)
{attribute 'hide'}
METHOD FB_init : BOOL
VAR_INPUT
	(*  if TRUE, the retain variables are initialized (warm start / cold start) *)
	bInitRetains : BOOL;
	(*  if TRUE, the instance afterwards gets moved into the copy code (online change) *)
	bInCopyCode : BOOL;
END_VAR
END_METHOD

{attribute 'TcTypeSystem'}

(* Internal method *)
{attribute 'hide'}
METHOD FB_exit : BOOL
VAR_INPUT
	(*  if TRUE, the exit method is called for exiting an instance that is copied afterwards (online change). *)
	bInCopyCode : BOOL;
END_VAR
END_METHOD

END_FUNCTION_BLOCK

// Synchronized Motion/MC_GearIn

{attribute 'c++_compatible'}
{attribute 'external_name' := 'MC_GearIn_GUID_D7A1F00E_B353_E326_E653_99E98F4ECC09'}
{attribute 'TcIecLibraryType'}
{attribute 'hide_all_locals'}
(* 
		This function block commands a ratio between the velocity of the slave and master axis.
	 *)
FUNCTION_BLOCK MC_GearIn
VAR_INPUT
	(* Reference to the master axis *)
	{attribute 'Namespace' := 'Tc3_Mc3Base'}
	Master : Tc3_Mc3Base.Type_Master1D;
	(* Reference to the slave axis *)
	{attribute 'GUID' := '931209B0-6FAC-E9BE-F824-23CE2FAA5732'}
	{attribute 'Namespace' := 'Tc3_Mc3Ptp'}
	Slave : REFERENCE TO AXIS_REF;
	(* Trigger the command with rising edge. *)
	Execute : BOOL;
END_VAR
VAR
	 {attribute 'hide'}
	_reserved1 : UINT_24_56;
END_VAR
VAR_INPUT
	(* Gear ratio numerator *)
	RatioNumerator : LREAL := 1.0;
	(* Gear ratio denominator *)
	RatioDenominator : UDINT := 1;
END_VAR
VAR
END_VAR
VAR_INPUT
	(* Maximum slave acceleration ([PosUnit]/s^2, positive) *)
	Acceleration : LREAL := STRING_TO_LREAL('#Default');
	(* Maximum slave deceleration ([PosUnit]/s^2, positive) *)
	Deceleration : LREAL := STRING_TO_LREAL('#Default');
	(* Maximum slave jerk ([PosUnit]/s^3, positive) *)
	Jerk : LREAL := STRING_TO_LREAL('#Default');
	(* Chronological sequence of the command *)
	{attribute 'Namespace' := 'Tc3_Mc3Base'}
	BufferMode : Tc3_Mc3Base.EBufferMode := Tc3_Mc3Base.EBufferMode.Aborting;
	(* Reaction if an error occurs in the master while this command is active. *)
	{attribute 'Namespace' := 'Tc3_Mc3Base'}
	ReactionToMasterError : Tc3_Mc3Base.EReactionToMasterError := Tc3_Mc3Base.EReactionToMasterError.TriggerSlaveError;
	(* Reaction if an error occurs in the slave while this command is active. *)
	{attribute 'Namespace' := 'Tc3_Mc3Base'}
	ReactionToSlaveError : Tc3_Mc3Base.EReactionToSlaveError := Tc3_Mc3Base.EReactionToSlaveError.TriggerMasterError;
END_VAR
VAR
END_VAR
VAR_OUTPUT
	(* Synchronization established *)
	InGear : BOOL;
	(* Function block is not finished and new output values are to be expected. *)
	Busy : BOOL;
	(* Function block has active control on the axis. *)
	Active : BOOL;
	(* Command is aborted by another command. *)
	CommandAborted : BOOL;
	(* Error occurred within function block. *)
	Error : BOOL;
END_VAR
VAR
	 {attribute 'hide'}
	_reserved2 : USINT;
END_VAR
VAR_OUTPUT
	(* Error identifier *)
	ErrorId : UDINT;
	(* Master is in error state. *)
	MasterHasError : BOOL;
END_VAR
VAR
	 {attribute 'hide'}
	_reserved3 : UINT_24_56;
	 {attribute 'hide'}
	_reserved4 : ARRAY [1..40] OF UINT_8_16;
	 {attribute 'hide'}
	_reserved5 : ARRAY [1..8] OF USINT;
END_VAR

{attribute 'TcTypeSystem'}

(* Internal method *)
{attribute 'hide'}
METHOD FB_init : BOOL
VAR_INPUT
	(*  if TRUE, the retain variables are initialized (warm start / cold start) *)
	bInitRetains : BOOL;
	(*  if TRUE, the instance afterwards gets moved into the copy code (online change) *)
	bInCopyCode : BOOL;
END_VAR
END_METHOD

{attribute 'TcTypeSystem'}

(* Internal method *)
{attribute 'hide'}
METHOD FB_exit : BOOL
VAR_INPUT
	(*  if TRUE, the exit method is called for exiting an instance that is copied afterwards (online change). *)
	bInCopyCode : BOOL;
END_VAR
END_METHOD

END_FUNCTION_BLOCK

// Synchronized Motion/MC_GearInPos

{attribute 'c++_compatible'}
{attribute 'pack_mode' := '1'}
{attribute 'external_name' := 'MC_GearInPos_GUID_4134C37A_5B73_E5EF_D747_25D272B58ACA'}
{attribute 'TcIecLibraryType'}
{attribute 'hide_all_locals'}
(* 
		This function block commands a gear ratio between the position of the slave and master axes
		from the synchronization point onwards.
	 *)
FUNCTION_BLOCK MC_GearInPos
VAR_INPUT
	(* Reference to the master axis *)
	{attribute 'Namespace' := 'Tc3_Mc3Base'}
	Master : Tc3_Mc3Base.Type_Master1D;
	(* Reference to the slave axis *)
	{attribute 'GUID' := '931209B0-6FAC-E9BE-F824-23CE2FAA5732'}
	{attribute 'Namespace' := 'Tc3_Mc3Ptp'}
	Slave : REFERENCE TO AXIS_REF;
	(* Trigger the command with rising edge. *)
	Execute : BOOL;
END_VAR
VAR
	 {attribute 'hide'}
	_reserved1 : UINT_24_56;
END_VAR
VAR_INPUT
	(* Gear ratio numerator *)
	RatioNumerator : LREAL := 1.0;
	(* Gear ratio denominator *)
	RatioDenominator : UDINT := 1;
END_VAR
VAR
	 {attribute 'hide'}
	_reserved2 : UDINT;
END_VAR
VAR_INPUT
	(* Position of master axis where master and slave axis are synchronized. *)
	MasterSyncPosition : LREAL := STRING_TO_LREAL('#Invalid');
	(* Position of slave axis where master and slave axis are synchronized. *)
	SlaveSyncPosition : LREAL := STRING_TO_LREAL('#Invalid');
	(* Maximum velocity during synchronization ([PosUnit]/s, positive) *)
	Velocity : LREAL := STRING_TO_LREAL('#Maximum');
	(* Maximum acceleration during synchronization ([PosUnit]/s^2, positive) *)
	Acceleration : LREAL := STRING_TO_LREAL('#Default');
	(* Maximum deceleration during synchronization ([PosUnit]/s^2, positive) *)
	Deceleration : LREAL := STRING_TO_LREAL('#Default');
	(* Maximum jerk during synchronization ([PosUnit]/s^3, positive) *)
	Jerk : LREAL := STRING_TO_LREAL('#Default');
	(* Chronological sequence of the command *)
	{attribute 'Namespace' := 'Tc3_Mc3Base'}
	BufferMode : Tc3_Mc3Base.EBufferMode := Tc3_Mc3Base.EBufferMode.Aborting;
	(* Reaction if an error occurs in the master while this command is active. *)
	{attribute 'Namespace' := 'Tc3_Mc3Base'}
	ReactionToMasterError : Tc3_Mc3Base.EReactionToMasterError := Tc3_Mc3Base.EReactionToMasterError.TriggerSlaveError;
	(* Reaction if an error occurs in the slave while this command is active. *)
	{attribute 'Namespace' := 'Tc3_Mc3Base'}
	ReactionToSlaveError : Tc3_Mc3Base.EReactionToSlaveError := Tc3_Mc3Base.EReactionToSlaveError.TriggerMasterError;
END_VAR
VAR
END_VAR
VAR_INPUT
	(* Allowed directions for establishing initial synchronization *)
	{attribute 'Namespace' := 'Tc3_Mc3Base'}
	AllowedSlaveSyncDirections : Tc3_Mc3Base.ESyncDirection := Tc3_Mc3Base.ESyncDirection.TowardsSlaveSyncPosition;
END_VAR
VAR
END_VAR
VAR_OUTPUT
	(* Synchronization started *)
	{attribute 'hide'}
	StartSync : BOOL;
	(* True if SyncState == InSync (slave coupled to the master AND master has passed its master sync position). *)
	InSync : BOOL;
END_VAR
VAR
	 {attribute 'hide'}
	_reserved3 : UINT;
END_VAR
VAR_OUTPUT
	(* Synchronization state. See EGearInPosSyncState for details. *)
	{attribute 'GUID' := 'C1F4A2D8-3B7E-4D5F-9A2C-8E6B1F0D4A93'}
	{attribute 'Namespace' := 'Tc3_Mc3Ptp'}
	SyncState : EGearInPosSyncState;
	(* Function block is not finished and new output values are to be expected. *)
	Busy : BOOL;
	(* Function block has active control on the axis. *)
	Active : BOOL;
	(* Command is aborted by another command. *)
	CommandAborted : BOOL;
	(* Error occurred within function block. *)
	Error : BOOL;
	(* Error identifier *)
	ErrorId : UDINT;
	(* Master is in error state. *)
	MasterHasError : BOOL;
END_VAR
VAR
	 {attribute 'hide'}
	_reserved4 : UINT_24_56;
	 {attribute 'hide'}
	_reserved5 : ARRAY [1..32] OF UINT_8_16;
	 {attribute 'hide'}
	_reserved6 : ARRAY [1..24] OF USINT;
END_VAR

{attribute 'TcTypeSystem'}

(* Internal method *)
{attribute 'hide'}
METHOD FB_init : BOOL
VAR_INPUT
	(*  if TRUE, the retain variables are initialized (warm start / cold start) *)
	bInitRetains : BOOL;
	(*  if TRUE, the instance afterwards gets moved into the copy code (online change) *)
	bInCopyCode : BOOL;
END_VAR
END_METHOD

{attribute 'TcTypeSystem'}

(* Internal method *)
{attribute 'hide'}
METHOD FB_exit : BOOL
VAR_INPUT
	(*  if TRUE, the exit method is called for exiting an instance that is copied afterwards (online change). *)
	bInCopyCode : BOOL;
END_VAR
END_METHOD

END_FUNCTION_BLOCK

// Administrative/MC_SetPosition

{attribute 'c++_compatible'}
{attribute 'external_name' := 'MC_SetPosition_GUID_14AA4E3B_998A_E180_F419_69B3FBB763F2'}
{attribute 'TcIecLibraryType'}
{attribute 'hide_all_locals'}
(* 
		This function block shifts the coordinate system of an axis by manipulating both the setpoint position as well as the
		actual position of an axis with the same value without any movement caused (Re-calibration with same following error).
		This can be used for instance for a reference situation.
	 *)
FUNCTION_BLOCK MC_SetPosition
VAR_INPUT
	(* Reference to the axis *)
	{attribute 'GUID' := 'F2078C57-FA2D-4316-A502-6E36DE58DC4A'}
	{attribute 'Namespace' := 'Tc3_Mc3Ptp'}
	Axis : Type_PtpSetPosition;
	(* Trigger the command with rising edge. *)
	Execute : BOOL;
END_VAR
VAR
	 {attribute 'hide'}
	_reserved1 : ARRAY [1..7] OF USINT;
END_VAR
VAR_INPUT
	(* New position value ([PosUnit]) or distance if Relative = TRUE *)
	Position : LREAL := STRING_TO_LREAL('#Invalid');
	(* Shift axis position by value *)
	Relative : BOOL := false;
	(* Resets position lag to zero. *)
	ClearPositionLag : BOOL;
END_VAR
VAR_OUTPUT
	(* Position has new value. *)
	Done : BOOL;
	(* Function block is not finished and new output values are to be expected. *)
	Busy : BOOL;
	(* Error occurred within function block. *)
	Error : BOOL;
END_VAR
VAR
	 {attribute 'hide'}
	_reserved2 : ARRAY [1..3] OF USINT;
END_VAR
VAR_OUTPUT
	(* Error identifier *)
	ErrorId : UDINT;
END_VAR
VAR
	 {attribute 'hide'}
	_reserved3 : UINT_0_32;
	 {attribute 'hide'}
	_reserved4 : ARRAY [1..20] OF UINT_8_16;
	 {attribute 'hide'}
	_reserved5 : ARRAY [1..32] OF USINT;
END_VAR

{attribute 'TcTypeSystem'}

(* Internal method *)
{attribute 'hide'}
METHOD FB_init : BOOL
VAR_INPUT
	(*  if TRUE, the retain variables are initialized (warm start / cold start) *)
	bInitRetains : BOOL;
	(*  if TRUE, the instance afterwards gets moved into the copy code (online change) *)
	bInCopyCode : BOOL;
END_VAR
END_METHOD

{attribute 'TcTypeSystem'}

(* Internal method *)
{attribute 'hide'}
METHOD FB_exit : BOOL
VAR_INPUT
	(*  if TRUE, the exit method is called for exiting an instance that is copied afterwards (online change). *)
	bInCopyCode : BOOL;
END_VAR
END_METHOD

END_FUNCTION_BLOCK

// External Setpoint Generator/MC_ActivateExternalSetpointGeneration

{attribute 'c++_compatible'}
{attribute 'external_name' := 'MC_ActivateExternalSetpointGeneration_GUID_F01B1D76_5347_ED41_C01F_C4347FBFE6A0'}
{attribute 'TcIecLibraryType'}
{attribute 'hide_all_locals'}
(* 
		This function block activates external setpoint generation.
		Setpoints are generated by a function block, which is called through the ITcMcExternalSetpointGenerator interface from the MC context.
		Additionally custom startup data can be passed through the generator.
	 *)
FUNCTION_BLOCK MC_ActivateExternalSetpointGeneration
VAR_IN_OUT
	(* Reference to the axis *)
	{attribute 'GUID' := '931209B0-6FAC-E9BE-F824-23CE2FAA5732'}
	{attribute 'Namespace' := 'Tc3_Mc3Ptp'}
	Axis : AXIS_REF;
END_VAR
VAR_INPUT
	(* Trigger the command with rising edge. *)
	Execute : BOOL;
END_VAR
VAR
	 {attribute 'hide'}
	_reserved1 : UINT_24_56;
END_VAR
VAR_INPUT
	(* Function block that implements (cyclic) methods for external setpoint generation *)
	{attribute 'GUID' := 'EF828E0B-69F0-4553-9DFF-4817D2FD6510'}
	ExternalSetpointGenerator : GLOBAL.ITcMcExternalSetpointGenerator;
	(* Allow the calling task to differ from the MC task (MET task). When TRUE, ensure compatible update rates and safe data access in the ITcMcExternalSetpointGenerator methods. *)
	AllowOtherContext : BOOL := false;
	(* Trigger error on inconsistent setpoint values (position, velocity, acceleration) if EnableDynamicChecks = TRUE. *)
	EnableDynamicChecks : BOOL := true;
END_VAR
VAR
	 {attribute 'hide'}
	_reserved2 : UINT_16_48;
END_VAR
VAR_INPUT
	(* Invocation identifier, passed through to the external setpoint generator. Can be used to distinguish multiple activations of the same generator, or to pass custom data (e.g. a pointer). *)
	{attribute 'GUID' := '18071995-0000-0000-0000-000000000073'}
	InvokeId : GLOBAL.XWORD := 0;
	(* Chronological sequence of the command *)
	{attribute 'Namespace' := 'Tc3_Mc3Base'}
	BufferMode : Tc3_Mc3Base.EBufferMode := Tc3_Mc3Base.EBufferMode.Aborting;
END_VAR
VAR_OUTPUT
	(* Function block is not finished and new output values are to be expected. *)
	Busy : BOOL;
	(* Function block has active control on the axis. *)
	Active : BOOL;
	(* Command is aborted by another command. *)
	CommandAborted : BOOL;
	(* Error occurred within function block. *)
	Error : BOOL;
END_VAR
VAR
	 {attribute 'hide'}
	_reserved3 : UINT;
END_VAR
VAR_OUTPUT
	(* Error identifier *)
	ErrorId : UDINT;
END_VAR
VAR
	 {attribute 'hide'}
	_reserved4 : UINT_0_32;
	 {attribute 'hide'}
	_reserved5 : ARRAY [1..32] OF UINT_8_16;
	 {attribute 'hide'}
	_reserved6 : ARRAY [1..24] OF USINT;
END_VAR

{attribute 'TcTypeSystem'}

(* Internal method *)
{attribute 'hide'}
METHOD FB_init : BOOL
VAR_INPUT
	(*  if TRUE, the retain variables are initialized (warm start / cold start) *)
	bInitRetains : BOOL;
	(*  if TRUE, the instance afterwards gets moved into the copy code (online change) *)
	bInCopyCode : BOOL;
END_VAR
END_METHOD

{attribute 'TcTypeSystem'}

(* Internal method *)
{attribute 'hide'}
METHOD FB_exit : BOOL
VAR_INPUT
	(*  if TRUE, the exit method is called for exiting an instance that is copied afterwards (online change). *)
	bInCopyCode : BOOL;
END_VAR
END_METHOD

END_FUNCTION_BLOCK

// External Setpoint Generator/MC_ExternalSetpointGenerator

{attribute 'c++_compatible'}
{attribute 'external_name' := 'MC_ExternalSetpointGenerator_GUID_395BF1E9_74A7_EC7E_CCDB_6EE07212C52C'}
{attribute 'TcIecLibraryType'}
{attribute 'no_explicit_call' :='do not call this POU directly'}
{attribute 'c++_compatible'}
{attribute 'hide_all_locals'}
(* 
	This function block provides the API to implement an external setpoint generator from the PLC environment.<br/>
The included callback methods are called from MC task context.<br/>
At least the OnCyclicSetpointGeneration method must be implemented.<br/>
<br/>
Requirements for deriving function block:<br/>
- The function block must implement ITcMcExternalSetpointGenerator interface.<br/>
- The function block and all overridden ITcMcExternalSetpointGenerator methods must have {attribute 'c++_compatible'}.<br/>
- The function block must override FB_init.<br/>
<br/>
Notes:<br/>
For online change compatibility the function block must have a FB_reinit method, in which MC_ExternalSetpointGenerator.FB_reinit() is called.
	 *)
FUNCTION_BLOCK ABSTRACT MC_ExternalSetpointGenerator IMPLEMENTS GLOBAL.ITComObject, GLOBAL.ITcMcExternalSetpointGenerator
VAR
	reserved : ARRAY [1..64] OF BYTE;
END_VAR

{attribute 'TcTypeSystem'}

(* (Internal method.) Initializes the function block with the object name. *)
METHOD FB_init : BOOL
VAR_INPUT
	(*  if TRUE, the retain variables are initialized (warm start / cold start) *)
	bInitRetains : BOOL;
	(*  if TRUE, the instance afterwards gets moved into the copy code (online change) *)
	bInCopyCode : BOOL;
	{attribute 'GUID' := '18071995-0000-0000-0000-000100000050'}
	sObjectName : STRING;
END_VAR
END_METHOD

{attribute 'TcTypeSystem'}

(* Internal method *)
METHOD FB_reinit : BOOL
END_METHOD

{attribute 'TcTypeSystem'}

(* Internal method *)
METHOD FB_exit : BOOL
VAR_INPUT
	(*  if TRUE, the exit method is called for exiting an instance that is copied afterwards (online change). *)
	bInCopyCode : BOOL;
END_VAR
END_METHOD

{attribute 'TcTypeSystem'}

(* Internal method *)
{attribute 'c++_compatible'}
{attribute 'hide'}
METHOD FINAL TcAddRef : UDINT
END_METHOD

{attribute 'TcTypeSystem'}

(* Internal method *)
{attribute 'c++_compatible'}
{attribute 'c++_external'}
{attribute 'hide'}
METHOD FINAL TcQueryInterface : GLOBAL.HRESULT
VAR_INPUT
	{attribute 'GUID' := '18071995-0000-0000-0000-000000000025'}
	iid : REFERENCE TO GLOBAL.IID;
	{attribute 'GUID' := '18071995-0000-0000-0000-000000000018'}
	pipItf : POINTER TO GLOBAL.PVOID;
END_VAR
END_METHOD

{attribute 'TcTypeSystem'}

(* Internal method *)
{attribute 'c++_compatible'}
{attribute 'c++_external'}
{attribute 'hide'}
METHOD FINAL TcRelease : UDINT
END_METHOD

{attribute 'TcTypeSystem'}

{attribute 'c++_compatible'}
{attribute 'c++_external'}
{attribute 'hide'}
METHOD FINAL GetClassId : GLOBAL.HRESULT
VAR_INPUT
	{attribute 'GUID' := '18071995-0000-0000-0000-000000000024'}
	classId : REFERENCE TO GLOBAL.CLSID;
END_VAR
END_METHOD

{attribute 'TcTypeSystem'}

{attribute 'c++_compatible'}
{attribute 'c++_external'}
{attribute 'hide'}
METHOD FINAL TcGetObjectId : GLOBAL.HRESULT
VAR_INPUT
	{attribute 'GUID' := '18071995-0000-0000-0000-00000000000F'}
	objId : REFERENCE TO GLOBAL.OTCID;
END_VAR
END_METHOD

{attribute 'TcTypeSystem'}

{attribute 'c++_compatible'}
{attribute 'c++_external'}
{attribute 'hide'}
METHOD FINAL TcGetObjectName : GLOBAL.HRESULT
VAR_INPUT
	objName : POINTER TO SINT;
	nameLen : UDINT;
END_VAR
END_METHOD

{attribute 'TcTypeSystem'}

{attribute 'c++_compatible'}
{attribute 'c++_external'}
{attribute 'hide'}
METHOD FINAL TcSetObjectId : GLOBAL.HRESULT
VAR_INPUT
	{attribute 'GUID' := '18071995-0000-0000-0000-00000000000F'}
	objId : GLOBAL.OTCID;
END_VAR
END_METHOD

{attribute 'TcTypeSystem'}

{attribute 'c++_compatible'}
{attribute 'c++_external'}
{attribute 'hide'}
METHOD FINAL TcSetObjectName : GLOBAL.HRESULT
VAR_INPUT
	objName : POINTER TO SINT;
END_VAR
END_METHOD

{attribute 'TcTypeSystem'}

{attribute 'c++_compatible'}
{attribute 'c++_external'}
{attribute 'hide'}
METHOD FINAL TcSetObjState : GLOBAL.HRESULT
VAR_INPUT
	{attribute 'GUID' := '18071995-0000-0000-0000-000000000061'}
	state : GLOBAL.TCOM_STATE;
	{attribute 'GUID' := '00000030-0000-0000-E000-000000000064'}
	ipSrv : GLOBAL.ITComObjectServer;
	{attribute 'GUID' := '8ADAFA6E-467B-49AA-BC54-CA235CC732A9'}
	pInitData : POINTER TO GLOBAL.TComInitDataHdr;
END_VAR
END_METHOD

{attribute 'TcTypeSystem'}

{attribute 'c++_compatible'}
{attribute 'c++_external'}
{attribute 'hide'}
METHOD FINAL TcGetObjState : GLOBAL.HRESULT
VAR_INPUT
	{attribute 'GUID' := '18071995-0000-0000-0000-000000000061'}
	pState : POINTER TO GLOBAL.TCOM_STATE;
END_VAR
END_METHOD

{attribute 'TcTypeSystem'}

{attribute 'c++_compatible'}
{attribute 'c++_external'}
{attribute 'hide'}
METHOD FINAL TcGetObjPara : GLOBAL.HRESULT
VAR_INPUT
	{attribute 'GUID' := '18071995-0000-0000-0000-00000000001C'}
	pid : GLOBAL.PTCID;
	nData : REFERENCE TO UDINT;
	{attribute 'GUID' := '18071995-0000-0000-0000-000000000018'}
	pData : REFERENCE TO GLOBAL.PVOID;
	{attribute 'GUID' := '18071995-0000-0000-0000-00000000001D'}
	pgp : GLOBAL.PTCGP := 0;
END_VAR
END_METHOD

{attribute 'TcTypeSystem'}

{attribute 'c++_compatible'}
{attribute 'c++_external'}
{attribute 'hide'}
METHOD FINAL TcSetObjPara : GLOBAL.HRESULT
VAR_INPUT
	{attribute 'GUID' := '18071995-0000-0000-0000-00000000001C'}
	pid : GLOBAL.PTCID;
	nData : UDINT;
	{attribute 'GUID' := '18071995-0000-0000-0000-000000000018'}
	pData : GLOBAL.PVOID;
	{attribute 'GUID' := '18071995-0000-0000-0000-00000000001D'}
	pgp : GLOBAL.PTCGP := 0;
END_VAR
END_METHOD

{attribute 'TcTypeSystem'}

{attribute 'c++_compatible'}
{attribute 'c++_external'}
{attribute 'hide'}
METHOD FINAL TcGetParentObjId : GLOBAL.HRESULT
VAR_INPUT
	{attribute 'GUID' := '18071995-0000-0000-0000-00000000000F'}
	objId : REFERENCE TO GLOBAL.OTCID;
END_VAR
END_METHOD

{attribute 'TcTypeSystem'}

{attribute 'c++_compatible'}
{attribute 'c++_external'}
{attribute 'hide'}
METHOD FINAL TcSetParentObjId : GLOBAL.HRESULT
VAR_INPUT
	{attribute 'GUID' := '18071995-0000-0000-0000-00000000000F'}
	objId : GLOBAL.OTCID;
END_VAR
END_METHOD

{attribute 'TcTypeSystem'}

(* Called once when the external setpoint generator is being prepared for activation. *)
{attribute 'c++_compatible'}
METHOD OnPreparation : GLOBAL.HRESULT
VAR_INPUT
	{attribute 'GUID' := '18071995-0000-0000-0000-000000000073'}
	InvokeId : GLOBAL.XWORD;
END_VAR
END_METHOD

{attribute 'TcTypeSystem'}

(* Called to initialize the starting point before cyclic setpoint generation begins. *)
{attribute 'c++_compatible'}
METHOD OnStartPointInitialization : GLOBAL.HRESULT
VAR_INPUT
	{attribute 'GUID' := '18071995-0000-0000-0000-000000000073'}
	InvokeId : GLOBAL.XWORD;
	StartDcTime : LINT;
	Position : LREAL;
	Velocity : LREAL;
	Acceleration : LREAL;
END_VAR
END_METHOD

{attribute 'TcTypeSystem'}

(* Called every MC cycle to compute the next setpoint values. Must be overridden. *)
{attribute 'c++_compatible'}
METHOD ABSTRACT OnCyclicSetpointGeneration : GLOBAL.HRESULT
VAR_INPUT
	{attribute 'GUID' := '18071995-0000-0000-0000-000000000073'}
	InvokeId : GLOBAL.XWORD;
	TimeInGeneration : LREAL;
	Position : REFERENCE TO LREAL;
	Velocity : REFERENCE TO LREAL;
	Acceleration : REFERENCE TO LREAL;
END_VAR
END_METHOD

{attribute 'TcTypeSystem'}

(* Called when the external setpoint generator is deactivated/aborted. *)
{attribute 'c++_compatible'}
METHOD OnDeactivation : GLOBAL.HRESULT
VAR_INPUT
	{attribute 'GUID' := '18071995-0000-0000-0000-000000000073'}
	InvokeId : GLOBAL.XWORD;
END_VAR
END_METHOD

END_FUNCTION_BLOCK

// Discrete Motion/MC_Halt

{attribute 'c++_compatible'}
{attribute 'external_name' := 'MC_Halt_GUID_AB802E1B_0B9F_EA95_F3F7_878827469A2D'}
{attribute 'TcIecLibraryType'}
{attribute 'hide_all_locals'}
(* 
		This function block commands a motion stop. The axis is transferred to the state DiscreteMotion, until
		zero dynamics is reached.
	 *)
FUNCTION_BLOCK MC_Halt
VAR_IN_OUT
	(* Reference to the axis *)
	{attribute 'GUID' := '931209B0-6FAC-E9BE-F824-23CE2FAA5732'}
	{attribute 'Namespace' := 'Tc3_Mc3Ptp'}
	Axis : AXIS_REF;
END_VAR
VAR_INPUT
	(* Trigger the command with rising edge. *)
	Execute : BOOL;
END_VAR
VAR
	 {attribute 'hide'}
	_reserved1 : ARRAY [1..7] OF USINT;
END_VAR
VAR_INPUT
	(* Maximum deceleration ([PosUnit]/s^2, positive) *)
	Deceleration : LREAL := STRING_TO_LREAL('#Default');
	(* Maximum jerk ([PosUnit]/s^3, positive) *)
	Jerk : LREAL := STRING_TO_LREAL('#Default');
END_VAR
VAR
	 {attribute 'hide'}
	_reserved2 : UINT;
END_VAR
VAR_OUTPUT
	(* Zero dynamics has been reached, axis state is transferred to Standstill. *)
	Done : BOOL;
	(* Function block is not finished and new output values are to be expected. *)
	Busy : BOOL;
	(* Function block has active control on the axis. *)
	Active : BOOL;
	(* Command is aborted by another command. *)
	CommandAborted : BOOL;
	(* Error occurred within function block. *)
	Error : BOOL;
END_VAR
VAR
	 {attribute 'hide'}
	_reserved3 : USINT;
END_VAR
VAR_OUTPUT
	(* Error identifier *)
	ErrorId : UDINT;
END_VAR
VAR
	 {attribute 'hide'}
	_reserved4 : UINT_0_32;
	 {attribute 'hide'}
	_reserved5 : ARRAY [1..28] OF UINT_8_16;
	 {attribute 'hide'}
	_reserved6 : ARRAY [1..32] OF USINT;
END_VAR

{attribute 'TcTypeSystem'}

(* Internal method *)
{attribute 'hide'}
METHOD FB_init : BOOL
VAR_INPUT
	(*  if TRUE, the retain variables are initialized (warm start / cold start) *)
	bInitRetains : BOOL;
	(*  if TRUE, the instance afterwards gets moved into the copy code (online change) *)
	bInCopyCode : BOOL;
END_VAR
END_METHOD

{attribute 'TcTypeSystem'}

(* Internal method *)
{attribute 'hide'}
METHOD FB_exit : BOOL
VAR_INPUT
	(*  if TRUE, the exit method is called for exiting an instance that is copied afterwards (online change). *)
	bInCopyCode : BOOL;
END_VAR
END_METHOD

END_FUNCTION_BLOCK

// Discrete Motion/MC_MoveAbsolute

{attribute 'c++_compatible'}
{attribute 'external_name' := 'MC_MoveAbsolute_GUID_7B11FF58_8031_EFF7_EA9C_E9F49CACCC6F'}
{attribute 'TcIecLibraryType'}
{attribute 'hide_all_locals'}
(* 
		This function block commands a motion to a specified absolute position.
	 *)
FUNCTION_BLOCK MC_MoveAbsolute
VAR_IN_OUT
	(* Reference to the axis *)
	{attribute 'GUID' := '931209B0-6FAC-E9BE-F824-23CE2FAA5732'}
	{attribute 'Namespace' := 'Tc3_Mc3Ptp'}
	Axis : AXIS_REF;
END_VAR
VAR_INPUT
	(* Trigger the command with rising edge. *)
	Execute : BOOL;
END_VAR
VAR
	 {attribute 'hide'}
	_reserved1 : ARRAY [1..7] OF USINT;
END_VAR
VAR_INPUT
	(* Commanded position ([PosUnit]) *)
	Position : LREAL := STRING_TO_LREAL('#Invalid');
	(* Maximum velocity ([PosUnit]/s, positive) *)
	Velocity : LREAL := STRING_TO_LREAL('#Invalid');
	(* Maximum acceleration ([PosUnit]/s^2, positive) *)
	Acceleration : LREAL := STRING_TO_LREAL('#Default');
	(* Maximum deceleration ([PosUnit]/s^2, positive) *)
	Deceleration : LREAL := STRING_TO_LREAL('#Default');
	(* Maximum jerk ([PosUnit]/s^3, positive) *)
	Jerk : LREAL := STRING_TO_LREAL('#Default');
	(* Chronological sequence of the command *)
	{attribute 'Namespace' := 'Tc3_Mc3Base'}
	BufferMode : Tc3_Mc3Base.EBufferMode := Tc3_Mc3Base.EBufferMode.Aborting;
END_VAR
VAR_OUTPUT
	(* Commanded position finally reached *)
	Done : BOOL;
	(* Function block is not finished and new output values are to be expected. *)
	Busy : BOOL;
	(* Function block has active control on the axis. *)
	Active : BOOL;
	(* Command is aborted by another command. *)
	CommandAborted : BOOL;
	(* Error occurred within function block. *)
	Error : BOOL;
END_VAR
VAR
	 {attribute 'hide'}
	_reserved2 : USINT;
END_VAR
VAR_OUTPUT
	(* Error identifier *)
	ErrorId : UDINT;
END_VAR
VAR
	 {attribute 'hide'}
	_reserved3 : UINT_0_32;
	 {attribute 'hide'}
	_reserved4 : ARRAY [1..36] OF UINT_8_16;
	 {attribute 'hide'}
	_reserved5 : ARRAY [1..16] OF USINT;
END_VAR

{attribute 'TcTypeSystem'}

(* Internal method *)
{attribute 'hide'}
METHOD FB_init : BOOL
VAR_INPUT
	(*  if TRUE, the retain variables are initialized (warm start / cold start) *)
	bInitRetains : BOOL;
	(*  if TRUE, the instance afterwards gets moved into the copy code (online change) *)
	bInCopyCode : BOOL;
END_VAR
END_METHOD

{attribute 'TcTypeSystem'}

(* Internal method *)
{attribute 'hide'}
METHOD FB_exit : BOOL
VAR_INPUT
	(*  if TRUE, the exit method is called for exiting an instance that is copied afterwards (online change). *)
	bInCopyCode : BOOL;
END_VAR
END_METHOD

END_FUNCTION_BLOCK

// Discrete Motion/MC_MoveModulo

{attribute 'c++_compatible'}
{attribute 'external_name' := 'MC_MoveModulo_GUID_8C793664_4941_EC4E_FF36_D6A623786731'}
{attribute 'TcIecLibraryType'}
{attribute 'hide_all_locals'}
(* 
		This function block commands a motion to a specified modulo position.
	 *)
FUNCTION_BLOCK MC_MoveModulo
VAR_IN_OUT
	(* Reference to the axis *)
	{attribute 'GUID' := '931209B0-6FAC-E9BE-F824-23CE2FAA5732'}
	{attribute 'Namespace' := 'Tc3_Mc3Ptp'}
	Axis : AXIS_REF;
END_VAR
VAR_INPUT
	(* Trigger the command with rising edge. *)
	Execute : BOOL;
END_VAR
VAR
	 {attribute 'hide'}
	_reserved1 : ARRAY [1..7] OF USINT;
END_VAR
VAR_INPUT
	(* Commanded modulo position ([PosUnit]) *)
	Position : LREAL := STRING_TO_LREAL('#Invalid');
	(* Number of additional modulo turns in the commanded direction. A value > 0 requires Direction <> EModuloDirection.ShortestDistance. *)
	AdditionalTurns : UDINT := 0;
END_VAR
VAR
	 {attribute 'hide'}
	_reserved2 : UDINT;
END_VAR
VAR_INPUT
	(* Maximum velocity ([PosUnit]/s, positive) *)
	Velocity : LREAL := STRING_TO_LREAL('#Invalid');
	(* Maximum acceleration ([PosUnit]/s^2, positive) *)
	Acceleration : LREAL := STRING_TO_LREAL('#Default');
	(* Maximum deceleration ([PosUnit]/s^2, positive) *)
	Deceleration : LREAL := STRING_TO_LREAL('#Default');
	(* Maximum jerk ([PosUnit]/s^3, positive) *)
	Jerk : LREAL := STRING_TO_LREAL('#Default');
	(* Chronological sequence of the command *)
	{attribute 'Namespace' := 'Tc3_Mc3Base'}
	BufferMode : Tc3_Mc3Base.EBufferMode := Tc3_Mc3Base.EBufferMode.Aborting;
	(* Commanded direction. Must have value <> EModuloDirection.ShortestDistance if AdditionalTurns has value > 0. *)
	{attribute 'GUID' := '1798FE53-EDB6-4788-B12C-B2244F2AA2F6'}
	{attribute 'Namespace' := 'Tc3_Mc3Ptp'}
	Direction : EModuloDirection := EModuloDirection.ShortestDistance;
END_VAR
VAR_OUTPUT
	(* Commanded position finally reached *)
	Done : BOOL;
	(* Function block is not finished and new output values are to be expected. *)
	Busy : BOOL;
	(* Function block has active control on the axis. *)
	Active : BOOL;
	(* Command is aborted by another command. *)
	CommandAborted : BOOL;
	(* Error occurred within function block. *)
	Error : BOOL;
END_VAR
VAR
	 {attribute 'hide'}
	_reserved3 : ARRAY [1..3] OF USINT;
END_VAR
VAR_OUTPUT
	(* Error identifier *)
	ErrorId : UDINT;
END_VAR
VAR
	 {attribute 'hide'}
	_reserved4 : UINT_0_32;
	 {attribute 'hide'}
	_reserved5 : ARRAY [1..36] OF UINT_8_16;
	 {attribute 'hide'}
	_reserved6 : ARRAY [1..12] OF USINT;
END_VAR

{attribute 'TcTypeSystem'}

(* Internal method *)
{attribute 'hide'}
METHOD FB_init : BOOL
VAR_INPUT
	(*  if TRUE, the retain variables are initialized (warm start / cold start) *)
	bInitRetains : BOOL;
	(*  if TRUE, the instance afterwards gets moved into the copy code (online change) *)
	bInCopyCode : BOOL;
END_VAR
END_METHOD

{attribute 'TcTypeSystem'}

(* Internal method *)
{attribute 'hide'}
METHOD FB_exit : BOOL
VAR_INPUT
	(*  if TRUE, the exit method is called for exiting an instance that is copied afterwards (online change). *)
	bInCopyCode : BOOL;
END_VAR
END_METHOD

END_FUNCTION_BLOCK

// Discrete Motion/MC_MoveRelative

{attribute 'c++_compatible'}
{attribute 'external_name' := 'MC_MoveRelative_GUID_554DD16A_33FF_EEAC_D66F_8AA7A5D0EA22'}
{attribute 'TcIecLibraryType'}
{attribute 'hide_all_locals'}
(* 
		This function block commands a motion of a specified distance relative
		to the set position at the time the command gets active.
	 *)
FUNCTION_BLOCK MC_MoveRelative
VAR_IN_OUT
	(* Reference to the axis *)
	{attribute 'GUID' := '931209B0-6FAC-E9BE-F824-23CE2FAA5732'}
	{attribute 'Namespace' := 'Tc3_Mc3Ptp'}
	Axis : AXIS_REF;
END_VAR
VAR_INPUT
	(* Trigger the command with rising edge. *)
	Execute : BOOL;
END_VAR
VAR
	 {attribute 'hide'}
	_reserved1 : ARRAY [1..7] OF USINT;
END_VAR
VAR_INPUT
	(* Relative distance ([PosUnit]) *)
	Distance : LREAL := STRING_TO_LREAL('#Invalid');
	(* Maximum velocity ([PosUnit]/s, positive) *)
	Velocity : LREAL := STRING_TO_LREAL('#Invalid');
	(* Maximum acceleration ([PosUnit]/s^2, positive) *)
	Acceleration : LREAL := STRING_TO_LREAL('#Default');
	(* Maximum deceleration ([PosUnit]/s^2, positive) *)
	Deceleration : LREAL := STRING_TO_LREAL('#Default');
	(* Maximum jerk ([PosUnit]/s^3, positive) *)
	Jerk : LREAL := STRING_TO_LREAL('#Default');
	(* Chronological sequence of the command *)
	{attribute 'Namespace' := 'Tc3_Mc3Base'}
	BufferMode : Tc3_Mc3Base.EBufferMode := Tc3_Mc3Base.EBufferMode.Aborting;
END_VAR
VAR_OUTPUT
	(* Commanded distance reached *)
	Done : BOOL;
	(* Function block is not finished and new output values are to be expected. *)
	Busy : BOOL;
	(* Function block has active control on the axis. *)
	Active : BOOL;
	(* Command is aborted by another command. *)
	CommandAborted : BOOL;
	(* Error occurred within function block. *)
	Error : BOOL;
END_VAR
VAR
	 {attribute 'hide'}
	_reserved2 : USINT;
END_VAR
VAR_OUTPUT
	(* Error identifier *)
	ErrorId : UDINT;
END_VAR
VAR
	 {attribute 'hide'}
	_reserved3 : UINT_0_32;
	 {attribute 'hide'}
	_reserved4 : ARRAY [1..28] OF UINT_8_16;
	 {attribute 'hide'}
	_reserved5 : ARRAY [1..32] OF USINT;
END_VAR

{attribute 'TcTypeSystem'}

(* Internal method *)
{attribute 'hide'}
METHOD FB_init : BOOL
VAR_INPUT
	(*  if TRUE, the retain variables are initialized (warm start / cold start) *)
	bInitRetains : BOOL;
	(*  if TRUE, the instance afterwards gets moved into the copy code (online change) *)
	bInCopyCode : BOOL;
END_VAR
END_METHOD

{attribute 'TcTypeSystem'}

(* Internal method *)
{attribute 'hide'}
METHOD FB_exit : BOOL
VAR_INPUT
	(*  if TRUE, the exit method is called for exiting an instance that is copied afterwards (online change). *)
	bInCopyCode : BOOL;
END_VAR
END_METHOD

END_FUNCTION_BLOCK

// Discrete Motion/MC_Stop

{attribute 'c++_compatible'}
{attribute 'external_name' := 'MC_Stop_GUID_0F8BAB3D_20CD_E2C6_C23C_95A0E4587BA1'}
{attribute 'TcIecLibraryType'}
{attribute 'hide_all_locals'}
(* 
		This function block commands a motion stop and transfers the axis to the state Stopping.
		It aborts any ongoing function block execution. While the axis is in state Stopping, no other function block can
		perform any motion on the same axis. The Done output is set immediately after zero dynamics is reached.
		The axis remains in the state Stopping as long as Execute is TRUE or zero dynamics is not yet reached. As
		soon as Done is SET and Execute is FALSE the axis goes to state Standstill.
	 *)
FUNCTION_BLOCK MC_Stop
VAR_IN_OUT
	(* Reference to the axis *)
	{attribute 'GUID' := '931209B0-6FAC-E9BE-F824-23CE2FAA5732'}
	{attribute 'Namespace' := 'Tc3_Mc3Ptp'}
	Axis : AXIS_REF;
END_VAR
VAR_INPUT
	(* Trigger the command with rising edge. While this is TRUE, other function blocks will be rejected for the axis. *)
	Execute : BOOL;
END_VAR
VAR
	 {attribute 'hide'}
	_reserved1 : ARRAY [1..7] OF USINT;
END_VAR
VAR_INPUT
	(* Maximum deceleration ([PosUnit]/s^2, positive) *)
	Deceleration : LREAL := STRING_TO_LREAL('#Default');
	(* Maximum jerk ([PosUnit]/s^3, positive) *)
	Jerk : LREAL := STRING_TO_LREAL('#Default');
END_VAR
VAR_OUTPUT
	(* Zero dynamics has been reached. *)
	Done : BOOL;
	(* Function block is not finished and new output values are to be expected. *)
	Busy : BOOL;
	(* Function block has active control on the axis. *)
	Active : BOOL;
	(* Command is aborted by another command. *)
	CommandAborted : BOOL;
	(* Error occurred within function block. *)
	Error : BOOL;
END_VAR
VAR
	 {attribute 'hide'}
	_reserved2 : ARRAY [1..3] OF USINT;
END_VAR
VAR_OUTPUT
	(* Error identifier *)
	ErrorId : UDINT;
END_VAR
VAR
	 {attribute 'hide'}
	_reserved3 : UINT_0_32;
	 {attribute 'hide'}
	_reserved4 : ARRAY [1..28] OF UINT_8_16;
	 {attribute 'hide'}
	_reserved5 : ARRAY [1..32] OF USINT;
END_VAR

{attribute 'TcTypeSystem'}

(* Internal method *)
{attribute 'hide'}
METHOD FB_init : BOOL
VAR_INPUT
	(*  if TRUE, the retain variables are initialized (warm start / cold start) *)
	bInitRetains : BOOL;
	(*  if TRUE, the instance afterwards gets moved into the copy code (online change) *)
	bInCopyCode : BOOL;
END_VAR
END_METHOD

{attribute 'TcTypeSystem'}

(* Internal method *)
{attribute 'hide'}
METHOD FB_exit : BOOL
VAR_INPUT
	(*  if TRUE, the exit method is called for exiting an instance that is copied afterwards (online change). *)
	bInCopyCode : BOOL;
END_VAR
END_METHOD

END_FUNCTION_BLOCK

// Discrete Motion/MC_WaitForStableActualPosition

{attribute 'c++_compatible'}
{attribute 'external_name' := 'MC_WaitForStableActualPosition_GUID_DBB75F0D_ED84_E00E_C719_EB8179A8A719'}
{attribute 'TcIecLibraryType'}
{attribute 'hide_all_locals'}
(* 
		This function block waits for a stable actual position.
		The command is always buffered and may only be triggered when the previous command ends with zero dynamics.
	 *)
FUNCTION_BLOCK MC_WaitForStableActualPosition
VAR_IN_OUT
	(* Reference to the axis *)
	{attribute 'GUID' := '931209B0-6FAC-E9BE-F824-23CE2FAA5732'}
	{attribute 'Namespace' := 'Tc3_Mc3Ptp'}
	Axis : AXIS_REF;
END_VAR
VAR_INPUT
	(* Trigger the command with rising edge. *)
	Execute : BOOL;
END_VAR
VAR
	 {attribute 'hide'}
	_reserved1 : ARRAY [1..7] OF USINT;
END_VAR
VAR_INPUT
	(* 
			Position tolerance around the set position ([PosUnit], positive). The actual position must remain within this window for the command to succeed.
		 *)
	PositionTolerance : LREAL := STRING_TO_LREAL('#Invalid');
	(* Duration (in seconds) that the actual position needs to consecutively stay inside the position window. Must have a value >= 0. *)
	WaitDuration : LREAL := STRING_TO_LREAL('#Invalid');
	(* 
			Duration (in seconds) after which an error is triggered if the actual position is not inside the position window.
			It can be left as 'Ignore' if no timeout is desired, otherwise must have a value > WaitDuration.
		 *)
	TimeoutDuration : LREAL := STRING_TO_LREAL('#Ignore');
END_VAR
VAR_OUTPUT
	(* Actual position is currently inside the position window. *)
	InPositionWindow : BOOL;
	(* Actual position has been consecutively inside the position window for at least WaitDuration. *)
	Done : BOOL;
	(* Function block is not finished and new output values are to be expected. *)
	Busy : BOOL;
	(* Function block has active control on the axis.
		While Active is TRUE, the set position remains on the final position
		of the previous command and the set dynamics remain zero. *)
	Active : BOOL;
	(* Command is aborted by another command. *)
	CommandAborted : BOOL;
	(* Error occurred within function block. *)
	Error : BOOL;
END_VAR
VAR
	 {attribute 'hide'}
	_reserved2 : UINT;
END_VAR
VAR_OUTPUT
	(* Error identifier *)
	ErrorId : UDINT;
END_VAR
VAR
	 {attribute 'hide'}
	_reserved3 : UINT_0_32;
	 {attribute 'hide'}
	_reserved4 : ARRAY [1..28] OF UINT_8_16;
	 {attribute 'hide'}
	_reserved5 : ARRAY [1..32] OF USINT;
END_VAR

{attribute 'TcTypeSystem'}

(* Internal method *)
{attribute 'hide'}
METHOD FB_init : BOOL
VAR_INPUT
	(*  if TRUE, the retain variables are initialized (warm start / cold start) *)
	bInitRetains : BOOL;
	(*  if TRUE, the instance afterwards gets moved into the copy code (online change) *)
	bInCopyCode : BOOL;
END_VAR
END_METHOD

{attribute 'TcTypeSystem'}

(* Internal method *)
{attribute 'hide'}
METHOD FB_exit : BOOL
VAR_INPUT
	(*  if TRUE, the exit method is called for exiting an instance that is copied afterwards (online change). *)
	bInCopyCode : BOOL;
END_VAR
END_METHOD

END_FUNCTION_BLOCK

// Synchronized Motion/MC_PhasingAbsolute

{attribute 'c++_compatible'}
{attribute 'external_name' := 'MC_PhasingAbsolute_GUID_0FB6BA3B_EE7E_E06E_EC12_68E5E404CC7B'}
{attribute 'TcIecLibraryType'}
{attribute 'hide_all_locals'}
(* 
		This function block commands an absolute phase shift in the master position of a synchronized slave axis.
		It is only valid for camming synchronization. The master axis is not aware of the phase shift.
	 *)
FUNCTION_BLOCK MC_PhasingAbsolute
VAR_INPUT
	(* Reference to the master axis *)
	{attribute 'Namespace' := 'Tc3_Mc3Base'}
	Master : Tc3_Mc3Base.Type_Master1D;
	(* Reference to the slave axis *)
	{attribute 'Namespace' := 'Tc3_Mc3Base'}
	Slave : Tc3_Mc3Base.Type_Phasing1D;
	(* Trigger the command with rising edge. *)
	Execute : BOOL;
END_VAR
VAR
	 {attribute 'hide'}
	_reserved1 : UINT_24_56;
END_VAR
VAR_INPUT
	(* Absolute phase difference in master position of the slave axis ([PosUnit]) *)
	PhaseShift : LREAL := STRING_TO_LREAL('#Invalid');
	(* Maximum velocity ([PosUnit]/s, positive) *)
	Velocity : LREAL := STRING_TO_LREAL('#Invalid');
	(* Maximum acceleration ([PosUnit]/s^2, positive) *)
	Acceleration : LREAL := STRING_TO_LREAL('#Invalid');
	(* Maximum deceleration ([PosUnit]/s^2, positive) *)
	Deceleration : LREAL := STRING_TO_LREAL('#Invalid');
	(* Maximum jerk ([PosUnit]/s^3, positive) *)
	Jerk : LREAL := STRING_TO_LREAL('#Invalid');
END_VAR
VAR_OUTPUT
	(* Commanded phasing reached *)
	Done : BOOL;
	(* Function block is not finished and new output values are to be expected. *)
	Busy : BOOL;
	(* Function block has active control on the axis. *)
	Active : BOOL;
	(* Command is aborted by another command. *)
	CommandAborted : BOOL;
	(* Error occurred within function block. *)
	Error : BOOL;
END_VAR
VAR
	 {attribute 'hide'}
	_reserved2 : ARRAY [1..3] OF USINT;
END_VAR
VAR_OUTPUT
	(* Error identifier *)
	ErrorId : UDINT;
END_VAR
VAR
	 {attribute 'hide'}
	_reserved3 : UDINT;
END_VAR
VAR_OUTPUT
	(* Current absolute phase shift between master and slave. *)
	AbsolutePhaseShift : LREAL;
END_VAR
VAR
	 {attribute 'hide'}
	_reserved4 : UINT_0_32;
	 {attribute 'hide'}
	_reserved5 : ARRAY [1..36] OF UINT_8_16;
	 {attribute 'hide'}
	_reserved6 : ARRAY [1..12] OF USINT;
END_VAR

{attribute 'TcTypeSystem'}

(* Internal method *)
{attribute 'hide'}
METHOD FB_init : BOOL
VAR_INPUT
	(*  if TRUE, the retain variables are initialized (warm start / cold start) *)
	bInitRetains : BOOL;
	(*  if TRUE, the instance afterwards gets moved into the copy code (online change) *)
	bInCopyCode : BOOL;
END_VAR
END_METHOD

{attribute 'TcTypeSystem'}

(* Internal method *)
{attribute 'hide'}
METHOD FB_exit : BOOL
VAR_INPUT
	(*  if TRUE, the exit method is called for exiting an instance that is copied afterwards (online change). *)
	bInCopyCode : BOOL;
END_VAR
END_METHOD

END_FUNCTION_BLOCK

// Synchronized Motion/MC_PhasingRelative

{attribute 'c++_compatible'}
{attribute 'external_name' := 'MC_PhasingRelative_GUID_9D2B4392_B836_E3CC_C617_FEDFC3194DB6'}
{attribute 'TcIecLibraryType'}
{attribute 'hide_all_locals'}
(* 
		This function block commands a relative phase shift in the master position of a synchronized slave axis.
		It is only valid for camming synchronization. The master axis is not aware of the phase shift.
	 *)
FUNCTION_BLOCK MC_PhasingRelative
VAR_INPUT
	(* Reference to the master axis *)
	{attribute 'Namespace' := 'Tc3_Mc3Base'}
	Master : Tc3_Mc3Base.Type_Master1D;
	(* Reference to the slave axis *)
	{attribute 'Namespace' := 'Tc3_Mc3Base'}
	Slave : Tc3_Mc3Base.Type_Phasing1D;
	(* Trigger the command with rising edge. *)
	Execute : BOOL;
END_VAR
VAR
	 {attribute 'hide'}
	_reserved1 : UINT_24_56;
END_VAR
VAR_INPUT
	(* Additional phase difference in master position of the slave axis ([PosUnit]) *)
	PhaseShift : LREAL := STRING_TO_LREAL('#Invalid');
	(* Maximum velocity ([PosUnit]/s, positive) *)
	Velocity : LREAL := STRING_TO_LREAL('#Invalid');
	(* Maximum acceleration ([PosUnit]/s^2, positive) *)
	Acceleration : LREAL := STRING_TO_LREAL('#Invalid');
	(* Maximum deceleration ([PosUnit]/s^2, positive) *)
	Deceleration : LREAL := STRING_TO_LREAL('#Invalid');
	(* Maximum jerk ([PosUnit]/s^3, positive) *)
	Jerk : LREAL := STRING_TO_LREAL('#Invalid');
END_VAR
VAR_OUTPUT
	(* Commanded phasing reached *)
	Done : BOOL;
	(* Function block is not finished and new output values are to be expected. *)
	Busy : BOOL;
	(* Function block has active control on the axis. *)
	Active : BOOL;
	(* Command is aborted by another command. *)
	CommandAborted : BOOL;
	(* Error occurred within function block. *)
	Error : BOOL;
END_VAR
VAR
	 {attribute 'hide'}
	_reserved2 : ARRAY [1..3] OF USINT;
END_VAR
VAR_OUTPUT
	(* Error identifier *)
	ErrorId : UDINT;
END_VAR
VAR
	 {attribute 'hide'}
	_reserved3 : UDINT;
END_VAR
VAR_OUTPUT
	(* Accumulated relative phase shift applied so far. *)
	CoveredPhaseShift : LREAL;
END_VAR
VAR
	 {attribute 'hide'}
	_reserved4 : UINT_0_32;
	 {attribute 'hide'}
	_reserved5 : ARRAY [1..36] OF UINT_8_16;
	 {attribute 'hide'}
	_reserved6 : ARRAY [1..12] OF USINT;
END_VAR

{attribute 'TcTypeSystem'}

(* Internal method *)
{attribute 'hide'}
METHOD FB_init : BOOL
VAR_INPUT
	(*  if TRUE, the retain variables are initialized (warm start / cold start) *)
	bInitRetains : BOOL;
	(*  if TRUE, the instance afterwards gets moved into the copy code (online change) *)
	bInCopyCode : BOOL;
END_VAR
END_METHOD

{attribute 'TcTypeSystem'}

(* Internal method *)
{attribute 'hide'}
METHOD FB_exit : BOOL
VAR_INPUT
	(*  if TRUE, the exit method is called for exiting an instance that is copied afterwards (online change). *)
	bInCopyCode : BOOL;
END_VAR
END_METHOD

END_FUNCTION_BLOCK

// Synchronized Motion/MC_HaltPhasing

{attribute 'c++_compatible'}
{attribute 'external_name' := 'MC_HaltPhasing_GUID_331FED17_F64A_E1C1_F7FE_BF15AC001F59'}
{attribute 'TcIecLibraryType'}
{attribute 'hide_all_locals'}
(* 
		This function block commands a phase shift stop in the master position of a synchronized slave axis.
		It is only valid for camming synchronization. The master axis is not aware of the phase shift.
	 *)
FUNCTION_BLOCK MC_HaltPhasing
VAR_INPUT
	(* Reference to the master axis *)
	{attribute 'Namespace' := 'Tc3_Mc3Base'}
	Master : Tc3_Mc3Base.Type_Master1D;
	(* Reference to the slave axis *)
	{attribute 'Namespace' := 'Tc3_Mc3Base'}
	Slave : Tc3_Mc3Base.Type_Phasing1D;
	(* Trigger the command with rising edge. *)
	Execute : BOOL;
END_VAR
VAR
	 {attribute 'hide'}
	_reserved1 : UINT_24_56;
END_VAR
VAR_INPUT
	(* Maximum deceleration ([PosUnit]/s^2, positive) *)
	Deceleration : LREAL := STRING_TO_LREAL('#Invalid');
	(* Maximum jerk ([PosUnit]/s^3, positive) *)
	Jerk : LREAL := STRING_TO_LREAL('#Invalid');
END_VAR
VAR_OUTPUT
	(* Zero dynamics has been reached, axis state is transferred to Standstill. *)
	Done : BOOL;
	(* Function block is not finished and new output values are to be expected. *)
	Busy : BOOL;
	(* Function block has active control on the axis. *)
	Active : BOOL;
	(* Command is aborted by another command. *)
	CommandAborted : BOOL;
	(* Error occurred within function block. *)
	Error : BOOL;
END_VAR
VAR
	 {attribute 'hide'}
	_reserved2 : ARRAY [1..3] OF USINT;
END_VAR
VAR_OUTPUT
	(* Error identifier *)
	ErrorId : UDINT;
END_VAR
VAR
	 {attribute 'hide'}
	_reserved3 : UINT_0_32;
	 {attribute 'hide'}
	_reserved4 : ARRAY [1..36] OF UINT_8_16;
	 {attribute 'hide'}
	_reserved5 : ARRAY [1..16] OF USINT;
END_VAR

{attribute 'TcTypeSystem'}

(* Internal method *)
{attribute 'hide'}
METHOD FB_init : BOOL
VAR_INPUT
	(*  if TRUE, the retain variables are initialized (warm start / cold start) *)
	bInitRetains : BOOL;
	(*  if TRUE, the instance afterwards gets moved into the copy code (online change) *)
	bInCopyCode : BOOL;
END_VAR
END_METHOD

{attribute 'TcTypeSystem'}

(* Internal method *)
{attribute 'hide'}
METHOD FB_exit : BOOL
VAR_INPUT
	(*  if TRUE, the exit method is called for exiting an instance that is copied afterwards (online change). *)
	bInCopyCode : BOOL;
END_VAR
END_METHOD

END_FUNCTION_BLOCK

// Continuous Motion/MC_MoveVelocity

{attribute 'c++_compatible'}
{attribute 'external_name' := 'MC_MoveVelocity_GUID_88051865_8DAC_E609_E2EE_D59E06F31E2B'}
{attribute 'TcIecLibraryType'}
{attribute 'hide_all_locals'}
(* 
		This function block commands an endless movement with a specified velocity.
	 *)
FUNCTION_BLOCK MC_MoveVelocity
VAR_IN_OUT
	(* Reference to the axis *)
	{attribute 'GUID' := '931209B0-6FAC-E9BE-F824-23CE2FAA5732'}
	{attribute 'Namespace' := 'Tc3_Mc3Ptp'}
	Axis : AXIS_REF;
END_VAR
VAR_INPUT
	(* Trigger the command with rising edge. *)
	Execute : BOOL;
END_VAR
VAR
	 {attribute 'hide'}
	_reserved1 : ARRAY [1..7] OF USINT;
END_VAR
VAR_INPUT
	(* Commanded velocity ([PosUnit]/s, the sign of this parameter determines the direction of movement). *)
	Velocity : LREAL := STRING_TO_LREAL('#Invalid');
	(* Maximum acceleration ([PosUnit]/s^2, positive) *)
	Acceleration : LREAL := STRING_TO_LREAL('#Default');
	(* Maximum deceleration ([PosUnit]/s^2, positive) *)
	Deceleration : LREAL := STRING_TO_LREAL('#Default');
	(* Maximum jerk ([PosUnit]/s^3, positive) *)
	Jerk : LREAL := STRING_TO_LREAL('#Default');
	(* Chronological sequence of the command *)
	{attribute 'Namespace' := 'Tc3_Mc3Base'}
	BufferMode : Tc3_Mc3Base.EBufferMode := Tc3_Mc3Base.EBufferMode.Aborting;
END_VAR
VAR_OUTPUT
	(* Commanded velocity reached *)
	InVelocity : BOOL;
	(* Function block is not finished and new output values are to be expected. *)
	Busy : BOOL;
	(* Function block has active control on the axis. *)
	Active : BOOL;
	(* Command is aborted by another command. *)
	CommandAborted : BOOL;
	(* Error occurred within function block. *)
	Error : BOOL;
END_VAR
VAR
	 {attribute 'hide'}
	_reserved2 : USINT;
END_VAR
VAR_OUTPUT
	(* Error identifier *)
	ErrorId : UDINT;
END_VAR
VAR
	 {attribute 'hide'}
	_reserved3 : UINT_0_32;
	 {attribute 'hide'}
	_reserved4 : ARRAY [1..12] OF UINT_8_16;
	 {attribute 'hide'}
	_reserved5 : ARRAY [1..64] OF USINT;
END_VAR

{attribute 'TcTypeSystem'}

(* Internal method *)
{attribute 'hide'}
METHOD FB_init : BOOL
VAR_INPUT
	(*  if TRUE, the retain variables are initialized (warm start / cold start) *)
	bInitRetains : BOOL;
	(*  if TRUE, the instance afterwards gets moved into the copy code (online change) *)
	bInCopyCode : BOOL;
END_VAR
END_METHOD

{attribute 'TcTypeSystem'}

(* Internal method *)
{attribute 'hide'}
METHOD FB_exit : BOOL
VAR_INPUT
	(*  if TRUE, the exit method is called for exiting an instance that is copied afterwards (online change). *)
	bInCopyCode : BOOL;
END_VAR
END_METHOD

END_FUNCTION_BLOCK

// Continuous Motion/MC_Jog

{attribute 'c++_compatible'}
{attribute 'external_name' := 'MC_Jog_GUID_A55F8027_C6D9_E5BF_EC56_16117212363C'}
{attribute 'TcIecLibraryType'}
{attribute 'hide_all_locals'}
(* 
		This function block enables an axis to be moved via manual keys in different modi.
	 *)
FUNCTION_BLOCK MC_Jog
VAR_IN_OUT
	(* Reference to the axis *)
	{attribute 'GUID' := '931209B0-6FAC-E9BE-F824-23CE2FAA5732'}
	{attribute 'Namespace' := 'Tc3_Mc3Ptp'}
	Axis : AXIS_REF;
END_VAR
VAR_INPUT
	(* The command is executed with a rising edge, and the axis is moved in positive direction.
		Depending on the mode, the axis moves as long as the signal remains TRUE,
		or it stops automatically after a specified distance. *)
	JogForward : BOOL;
	(* The command is executed with a rising edge, and the axis is moved in negative direction.
		Depending on the mode, the axis moves as long as the signal remains TRUE,
		or it stops automatically after a specified distance. *)
	JogBackward : BOOL;
	(* Determines the operation mode in which the manual function is executed. *)
	{attribute 'GUID' := '81AB5A5F-F1B6-4D6D-83FB-05EE8E17A103'}
	{attribute 'Namespace' := 'Tc3_Mc3Ptp'}
	Mode : EJogMode := EJogMode.StandardSlow;
END_VAR
VAR
	 {attribute 'hide'}
	_reserved1 : UDINT;
END_VAR
VAR_INPUT
	(* Distance for movements in Mode Inching *)
	Distance : LREAL := STRING_TO_LREAL('#Ignore');
	(* Jog velocity ([PosUnit]/s, positive). Required for Continuous and Inching modes; StandardSlow and StandardFast use axis defaults. *)
	Velocity : LREAL := STRING_TO_LREAL('#Ignore');
	(* Maximum acceleration ([PosUnit]/s^2, positive) *)
	Acceleration : LREAL := STRING_TO_LREAL('#Default');
	(* Maximum deceleration ([PosUnit]/s^2, positive) *)
	Deceleration : LREAL := STRING_TO_LREAL('#Default');
	(* Maximum jerk ([PosUnit]/s^3, positive) *)
	Jerk : LREAL := STRING_TO_LREAL('#Default');
END_VAR
VAR_OUTPUT
	(* Function block has succeeded. *)
	Done : BOOL;
	(* Function block is not finished and new output values are to be expected. *)
	Busy : BOOL;
	(* Function block has active control on the axis. *)
	Active : BOOL;
	(* Command is aborted by another command. *)
	CommandAborted : BOOL;
	(* Error occurred within function block. *)
	Error : BOOL;
END_VAR
VAR
	 {attribute 'hide'}
	_reserved2 : ARRAY [1..3] OF USINT;
END_VAR
VAR_OUTPUT
	(* Error identifier *)
	ErrorId : UDINT;
END_VAR
VAR
	 {attribute 'hide'}
	_reserved3 : UINT_0_32;
	 {attribute 'hide'}
	_reserved4 : ARRAY [1..116] OF UINT_8_16;
	 {attribute 'hide'}
	_reserved5 : ARRAY [1..336] OF USINT;
END_VAR

{attribute 'TcTypeSystem'}

(* Internal method *)
{attribute 'hide'}
METHOD FB_init : BOOL
VAR_INPUT
	(*  if TRUE, the retain variables are initialized (warm start / cold start) *)
	bInitRetains : BOOL;
	(*  if TRUE, the instance afterwards gets moved into the copy code (online change) *)
	bInCopyCode : BOOL;
END_VAR
END_METHOD

{attribute 'TcTypeSystem'}

(* Internal method *)
{attribute 'hide'}
METHOD FB_exit : BOOL
VAR_INPUT
	(*  if TRUE, the exit method is called for exiting an instance that is copied afterwards (online change). *)
	bInCopyCode : BOOL;
END_VAR
END_METHOD

END_FUNCTION_BLOCK

// Homing/MC_SetHomingState

{attribute 'c++_compatible'}
{attribute 'external_name' := 'MC_SetHomingState_GUID_3184677B_E360_EDB9_F0DA_83A3BDA06689'}
{attribute 'TcIecLibraryType'}
{attribute 'hide_all_locals'}
(* 
		This function block allows setting and resetting the IsPositionValid flag in the CDT_MCTOPLC_AXIS_STD. Optionally, it can also set the Position. 
	 *)
FUNCTION_BLOCK MC_SetHomingState
VAR_INPUT
	(* Reference to the axis *)
	{attribute 'GUID' := 'D4E5F6A7-B8C9-4D0E-1F2A-3B4C5D6E7F80'}
	{attribute 'Namespace' := 'Tc3_Mc3Ptp'}
	Axis : Type_PtpSetHomingState;
	(* Trigger the command with rising edge. *)
	Execute : BOOL;
END_VAR
VAR
	 {attribute 'hide'}
	_reserved1 : ARRAY [1..7] OF USINT;
END_VAR
VAR_INPUT
	(* New position value ([PosUnit]) *)
	Position : LREAL := STRING_TO_LREAL('#Invalid');
	(* Homing mode selection *)
	{attribute 'GUID' := 'EF80436F-EB50-4932-9829-D962EB4481D6'}
	{attribute 'Namespace' := 'Tc3_Mc3Ptp'}
	Mode : EHomingMode := EHomingMode.ForceIsHomed;
END_VAR
VAR_OUTPUT
	(* Homing succeeded *)
	Done : BOOL;
	(* Function block is not finished and new output values are to be expected. *)
	Busy : BOOL;
	(* Function block has active control on the axis. *)
	Active : BOOL;
	(* Command is aborted by another command. *)
	CommandAborted : BOOL;
	(* Error occurred within function block. *)
	Error : BOOL;
END_VAR
VAR
	 {attribute 'hide'}
	_reserved2 : ARRAY [1..3] OF USINT;
END_VAR
VAR_OUTPUT
	(* Error identifier *)
	ErrorId : UDINT;
END_VAR
VAR
	 {attribute 'hide'}
	_reserved3 : UINT_0_32;
	 {attribute 'hide'}
	_reserved4 : ARRAY [1..36] OF UINT_8_16;
	 {attribute 'hide'}
	_reserved5 : ARRAY [1..12] OF USINT;
END_VAR

{attribute 'TcTypeSystem'}

(* Internal method *)
{attribute 'hide'}
METHOD FB_init : BOOL
VAR_INPUT
	(*  if TRUE, the retain variables are initialized (warm start / cold start) *)
	bInitRetains : BOOL;
	(*  if TRUE, the instance afterwards gets moved into the copy code (online change) *)
	bInCopyCode : BOOL;
END_VAR
END_METHOD

{attribute 'TcTypeSystem'}

(* Internal method *)
{attribute 'hide'}
METHOD FB_exit : BOOL
VAR_INPUT
	(*  if TRUE, the exit method is called for exiting an instance that is copied afterwards (online change). *)
	bInCopyCode : BOOL;
END_VAR
END_METHOD

END_FUNCTION_BLOCK

// Homing/MC_Home

{attribute 'c++_compatible'}
{attribute 'external_name' := 'MC_Home_GUID_14031A25_D89E_E47F_F6DE_924E764254BA'}
{attribute 'TcIecLibraryType'}
{attribute 'hide_all_locals'}
(* 
		This function block commands the axis to perform the homing sequence.
		The homing sequence is added via the homing TCOM object.
		The calculated offset is stored in 'Active Homing Offset'.
		Offsets from MC_SetPosition are discarded.
	 *)
FUNCTION_BLOCK MC_Home
VAR_IN_OUT
	(* Reference to the axis *)
	{attribute 'GUID' := '931209B0-6FAC-E9BE-F824-23CE2FAA5732'}
	{attribute 'Namespace' := 'Tc3_Mc3Ptp'}
	Axis : AXIS_REF;
END_VAR
VAR_INPUT
	(* Trigger the command with rising edge. *)
	Execute : BOOL;
END_VAR
VAR
	 {attribute 'hide'}
	_reserved1 : ARRAY [1..7] OF USINT;
END_VAR
VAR_INPUT
	(* Absolute position at the reference signal ([PosUnit]) *)
	Position : LREAL := STRING_TO_LREAL('#Default');
END_VAR
VAR_OUTPUT
	(* 'Search home' sequence succeeded *)
	Done : BOOL;
	(* Function block is not finished and new output values are to be expected. *)
	Busy : BOOL;
	(* Function block has active control on the axis. *)
	Active : BOOL;
	(* Command is aborted by another command. *)
	CommandAborted : BOOL;
	(* Error occurred within function block. *)
	Error : BOOL;
END_VAR
VAR
	 {attribute 'hide'}
	_reserved2 : ARRAY [1..3] OF USINT;
END_VAR
VAR_OUTPUT
	(* Error identifier *)
	ErrorId : UDINT;
END_VAR
VAR
	 {attribute 'hide'}
	_reserved3 : UINT_0_32;
	 {attribute 'hide'}
	_reserved4 : ARRAY [1..28] OF UINT_8_16;
	 {attribute 'hide'}
	_reserved5 : ARRAY [1..32] OF USINT;
END_VAR

{attribute 'TcTypeSystem'}

(* Internal method *)
{attribute 'hide'}
METHOD FB_init : BOOL
VAR_INPUT
	(*  if TRUE, the retain variables are initialized (warm start / cold start) *)
	bInitRetains : BOOL;
	(*  if TRUE, the instance afterwards gets moved into the copy code (online change) *)
	bInCopyCode : BOOL;
END_VAR
END_METHOD

{attribute 'TcTypeSystem'}

(* Internal method *)
{attribute 'hide'}
METHOD FB_exit : BOOL
VAR_INPUT
	(*  if TRUE, the exit method is called for exiting an instance that is copied afterwards (online change). *)
	bInCopyCode : BOOL;
END_VAR
END_METHOD

END_FUNCTION_BLOCK

// TouchProbe/MC_TouchProbe

{attribute 'c++_compatible'}
{attribute 'external_name' := 'MC_TouchProbe_GUID_0BF8BF65_C83E_E4ED_C65A_A6F86A1DCED2'}
{attribute 'TcIecLibraryType'}
{attribute 'hide_all_locals'}
(* 
		This function block controls the recording of an axis position at a trigger event.<br/>
		One of WindowFirstPosition or WindowLastPosition can be left as 'Ignore' if no corresponding limit is desired.
	 *)
FUNCTION_BLOCK MC_TouchProbe
VAR
END_VAR
VAR_INPUT
	(* Reference to the axis *)
	{attribute 'GUID' := 'C7A9D3E5-6B1F-4E82-9C14-7D82F5A0B3E2'}
	{attribute 'Namespace' := 'Tc3_Mc3Ptp'}
	Axis : Type_PtpTouchProbe;
END_VAR
VAR
END_VAR
VAR_IN_OUT
	(* Reference to the trigger signal source like DriveTouchProbeRef or BinaryTouchProbeRef *)
	{attribute 'GUID' := 'CC3262A1-A7A1-46D3-802E-9117404E77E7'}
	{attribute 'Namespace' := 'Tc3_Mc3Ptp'}
	TriggerInput : TRIGGER_REF;
END_VAR
VAR
END_VAR
VAR_INPUT
	(* Trigger the command with rising edge. *)
	Execute : BOOL;
END_VAR
VAR
	 {attribute 'hide'}
	_reserved1 : ARRAY [1..7] OF USINT;
END_VAR
VAR_INPUT
	(* Options for the touch probe *)
	{attribute 'GUID' := 'F9D597B1-6D34-4DD9-A264-FACE1E14FDB6'}
	{attribute 'Namespace' := 'Tc3_Mc3Ptp'}
	Options : TouchProbeOptions;
END_VAR
VAR_OUTPUT
	(* Touch probe process succeeded *)
	Done : BOOL;
	(* Function block is not finished and new output values are to be expected. *)
	Busy : BOOL;
	(* Command is aborted by another command (MC_AbortTrigger). *)
	CommandAborted : BOOL;
	(* Error occurred within function block. *)
	Error : BOOL;
	(* Error identifier *)
	ErrorId : UDINT;
	(* Position where trigger event occurred ([PosUnit]). *)
	RecordedPosition : LREAL;
	(* DcTime at trigger event *)
	RecordedDcTimestamp : LINT;
	(* Number of recorded trigger events *)
	RecordedEventCounter : UDINT;
	(* TRUE if the recorded position is within the configured window. *)
	InWindow : BOOL;
END_VAR
VAR
	 {attribute 'hide'}
	_reserved2 : ARRAY [1..91] OF USINT;
END_VAR

{attribute 'TcTypeSystem'}

(* Internal method *)
{attribute 'hide'}
METHOD FB_init : BOOL
VAR_INPUT
	(*  if TRUE, the retain variables are initialized (warm start / cold start) *)
	bInitRetains : BOOL;
	(*  if TRUE, the instance afterwards gets moved into the copy code (online change) *)
	bInCopyCode : BOOL;
END_VAR
END_METHOD

{attribute 'TcTypeSystem'}

(* Internal method *)
{attribute 'hide'}
METHOD FB_exit : BOOL
VAR_INPUT
	(*  if TRUE, the exit method is called for exiting an instance that is copied afterwards (online change). *)
	bInCopyCode : BOOL;
END_VAR
END_METHOD

END_FUNCTION_BLOCK

// TouchProbe/DriveTouchProbeRef

{attribute 'c++_compatible'}
{attribute 'external_name' := 'DriveTouchProbeRef_GUID_FBFB08F3_8469_EFDD_C0F1_672E54CB6634'}
{attribute 'TcIecLibraryType'}
{attribute 'no_explicit_call' :='do not call this POU directly'}
{attribute 'no_assign_warning'}
(* TouchProbeRef for Drive Touch Probe. *)
FUNCTION_BLOCK DriveTouchProbeRef
VAR
END_VAR
VAR_INPUT
	(* Drive Settings *)
	{attribute 'GUID' := '6CD9C878-CAE9-4648-82CF-CD223730B518'}
	{attribute 'Namespace' := 'Tc3_Mc3Ptp'}
	CoeDriveSettings : CoeTouchProbeSettings;
END_VAR
VAR_OUTPUT
	(* Connect to MC_Touchprobe/MC_AbortTrigger TriggerInput *)
	{attribute 'GUID' := '0A344DB1-12B6-41C7-A8E3-C1B73FE15631'}
	{attribute 'Namespace' := 'Tc3_Mc3Ptp'}
	TouchProbe1 : TouchProbeUnit;
	(* Connect to MC_Touchprobe/MC_AbortTrigger TriggerInput *)
	{attribute 'GUID' := '0A344DB1-12B6-41C7-A8E3-C1B73FE15631'}
	{attribute 'Namespace' := 'Tc3_Mc3Ptp'}
	TouchProbe2 : TouchProbeUnit;
END_VAR
VAR
	 {attribute 'hide'}
	_reserved1 : ARRAY [1..8] OF USINT;
END_VAR

{attribute 'TcTypeSystem'}

(* Internal method *)
{attribute 'hide'}
METHOD FB_init : BOOL
VAR_INPUT
	(*  if TRUE, the retain variables are initialized (warm start / cold start) *)
	bInitRetains : BOOL;
	(*  if TRUE, the instance afterwards gets moved into the copy code (online change) *)
	bInCopyCode : BOOL;
END_VAR
END_METHOD

{attribute 'TcTypeSystem'}

(* Internal method *)
{attribute 'hide'}
METHOD FB_reinit : BOOL
END_METHOD

{attribute 'TcTypeSystem'}

(* Internal method *)
{attribute 'hide'}
METHOD FB_exit : BOOL
VAR_INPUT
	(*  if TRUE, the exit method is called for exiting an instance that is copied afterwards (online change). *)
	bInCopyCode : BOOL;
END_VAR
END_METHOD

END_FUNCTION_BLOCK

// TouchProbe/MC_AbortTrigger

{attribute 'c++_compatible'}
{attribute 'external_name' := 'MC_AbortTrigger_GUID_BF8E4F78_F7BC_E9C3_FCAD_14D9C3DBECA3'}
{attribute 'TcIecLibraryType'}
{attribute 'hide_all_locals'}
(* 
		This Function Block is used to abort function blocks which are used to record trigger events (e.g. MC_TouchProbe).
	 *)
FUNCTION_BLOCK MC_AbortTrigger
VAR
END_VAR
VAR_INPUT
	(* Reference to the axis *)
	{attribute 'GUID' := 'C7A9D3E5-6B1F-4E82-9C14-7D82F5A0B3E2'}
	{attribute 'Namespace' := 'Tc3_Mc3Ptp'}
	Axis : Type_PtpTouchProbe;
END_VAR
VAR
END_VAR
VAR_IN_OUT
	(* Reference to the trigger signal source like DriveTouchProbeRef or BinaryTouchProbeRef *)
	{attribute 'GUID' := 'CC3262A1-A7A1-46D3-802E-9117404E77E7'}
	{attribute 'Namespace' := 'Tc3_Mc3Ptp'}
	TriggerInput : TRIGGER_REF;
END_VAR
VAR
END_VAR
VAR_INPUT
	(* Aborts the monitoring of trigger event at rising edge. *)
	Execute : BOOL;
END_VAR
VAR_OUTPUT
	(* Abort Trigger succeeded *)
	Done : BOOL;
	(* Function block is not finished and new output values are to be expected. *)
	Busy : BOOL;
	(* Error occurred within function block. *)
	Error : BOOL;
	(* Error identifier *)
	ErrorId : UDINT;
END_VAR
VAR
	 {attribute 'hide'}
	_reserved1 : ARRAY [1..88] OF USINT;
END_VAR

{attribute 'TcTypeSystem'}

(* Internal method *)
{attribute 'hide'}
METHOD FB_init : BOOL
VAR_INPUT
	(*  if TRUE, the retain variables are initialized (warm start / cold start) *)
	bInitRetains : BOOL;
	(*  if TRUE, the instance afterwards gets moved into the copy code (online change) *)
	bInCopyCode : BOOL;
END_VAR
END_METHOD

{attribute 'TcTypeSystem'}

(* Internal method *)
{attribute 'hide'}
METHOD FB_exit : BOOL
VAR_INPUT
	(*  if TRUE, the exit method is called for exiting an instance that is copied afterwards (online change). *)
	bInCopyCode : BOOL;
END_VAR
END_METHOD

END_FUNCTION_BLOCK

// TouchProbe/BinaryTouchProbeRef

{attribute 'c++_compatible'}
{attribute 'external_name' := 'BinaryTouchProbeRef_GUID_26A9CC97_F97E_E3BD_E972_BA19B2A447C1'}
{attribute 'TcIecLibraryType'}
{attribute 'no_explicit_call' :='do not call this POU directly'}
{attribute 'no_assign_warning'}
(* TouchProbeRef for Binary Touch Probes. *)
FUNCTION_BLOCK BinaryTouchProbeRef
VAR
END_VAR
VAR_INPUT
	(* Link to Axis Touch Probe Object -> Oid. *)
	{attribute 'GUID' := '18071995-0000-0000-0000-00000000000F'}
	Oid AT %I* : GLOBAL.OTCID;
END_VAR
VAR
	 {attribute 'hide'}
	_reserved1 : UDINT;
END_VAR
VAR_OUTPUT
	(* Connect to MC_Touchprobe/MC_AbortTrigger TriggerInput *)
	{attribute 'GUID' := '0A344DB1-12B6-41C7-A8E3-C1B73FE15631'}
	{attribute 'Namespace' := 'Tc3_Mc3Ptp'}
	TouchProbe : TouchProbeUnit;
END_VAR

{attribute 'TcTypeSystem'}

(* Internal method *)
{attribute 'hide'}
METHOD FB_init : BOOL
VAR_INPUT
	(*  if TRUE, the retain variables are initialized (warm start / cold start) *)
	bInitRetains : BOOL;
	(*  if TRUE, the instance afterwards gets moved into the copy code (online change) *)
	bInCopyCode : BOOL;
END_VAR
END_METHOD

{attribute 'TcTypeSystem'}

(* Internal method *)
{attribute 'hide'}
METHOD FB_reinit : BOOL
END_METHOD

{attribute 'TcTypeSystem'}

(* Internal method *)
{attribute 'hide'}
METHOD FB_exit : BOOL
VAR_INPUT
	(*  if TRUE, the exit method is called for exiting an instance that is copied afterwards (online change). *)
	bInCopyCode : BOOL;
END_VAR
END_METHOD

END_FUNCTION_BLOCK

// TouchProbe/EncoderTouchProbeRef

